KUKA KRL program: MyProgram_139().src

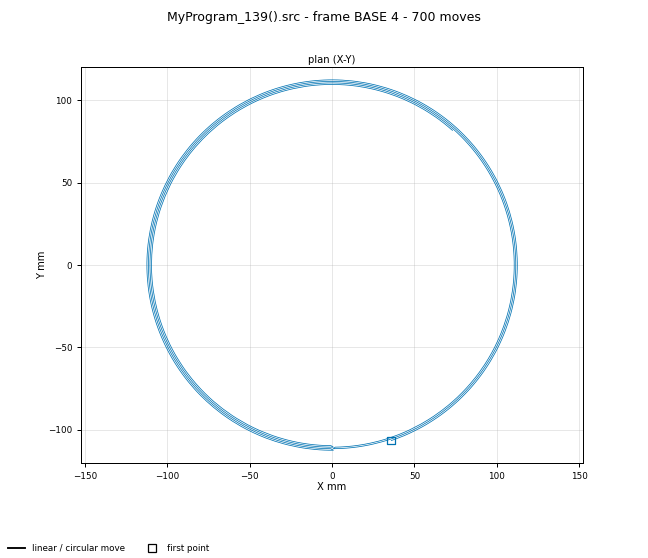
[picture p0: tool path of MyProgram_139().src in frame BASE 4, 700 of 700 moves have a stored position in this frame; points joined in program order, loops and branches not executed]
&ACCESS RVP
&REL 1
&PARAM TEMPLATE = C:\KRC\Roboter\Template\vorgabe
&PARAM EDITMASK = *
DEF MyProgram_139()
; ---- Setting reference (Base) ----
$BASE = BASE_DATA[4]

; --------------------------
; ---- Setting tool (TCP) ----
$TOOL = TOOL_DATA[3]
; --------------------------

$VEL.CP = VEL_APROX_PRINT
Startdeposition()
$VEL.CP = VEL_PRINT
LIN {X 35.9245,Y -106.4874,Z 112,A -74.797,B 24.9523,C -1.5971,E1 25.0523,E2 520.6725} C_DIS
LIN {X 38.4921,Y -105.5865,Z 112,A -73.3956,B 24.9521,C -1.5996,E1 25.056,E2 519.2681} C_DIS
LIN {X 41.1063,Y -104.5964,Z 112,A -71.9841,B 24.952,C -1.6009,E1 25.0597,E2 517.8564} C_DIS
LIN {X 43.6266,Y -103.5706,Z 112,A -70.5551,B 24.9517,C -1.6048,E1 25.0634,E2 516.4215} C_DIS
LIN {X 46.9304,Y -102.1175,Z 112,A -68.8328,B 24.9519,C -1.6024,E1 25.0677,E2 514.7093} C_DIS
LIN {X 49.2943,Y -100.9985,Z 112,A -67.3119,B 24.9513,C -1.6129,E1 25.0716,E2 513.1676} C_DIS
LIN {X 51.7581,Y -99.7583,Z 112,A -66.037,B 24.9515,C -1.6094,E1 25.0748,E2 511.9044} C_DIS
LIN {X 54.1907,Y -98.458,Z 112,A -64.636,B 24.9513,C -1.6116,E1 25.0782,E2 510.5022} C_DIS
LIN {X 56.5907,Y -97.0985,Z 112,A -63.2354,B 24.9512,C -1.6139,E1 25.0816,E2 509.1003} C_DIS
LIN {X 58.9565,Y -95.6804,Z 112,A -61.8347,B 24.951,C -1.6163,E1 25.0849,E2 507.6984} C_DIS
LIN {X 61.2869,Y -94.2047,Z 112,A -60.4345,B 24.9509,C -1.6188,E1 25.0882,E2 506.2969} C_DIS
LIN {X 63.5803,Y -92.6723,Z 112,A -59.034,B 24.9507,C -1.6214,E1 25.0915,E2 504.8951} C_DIS
LIN {X 65.8355,Y -91.0841,Z 112,A -57.6342,B 24.9506,C -1.624,E1 25.0947,E2 503.4939} C_DIS
LIN {X 68.051,Y -89.4409,Z 112,A -56.2343,B 24.9504,C -1.6267,E1 25.0978,E2 502.0926} C_DIS
LIN {X 70.2255,Y -87.744,Z 112,A -54.8346,B 24.9502,C -1.6295,E1 25.1009,E2 500.6916} C_DIS
LIN {X 72.7084,Y -85.6953,Z 112,A -53.1456,B 24.9499,C -1.6354,E1 25.1045,E2 498.995} C_DIS
LIN {X 74.9462,Y -83.7449,Z 112,A -51.6871,B 24.9499,C -1.6364,E1 25.1075,E2 497.54} C_DIS
LIN {X 76.9788,Y -81.8804,Z 112,A -50.292,B 24.9496,C -1.6393,E1 25.1104,E2 496.1439} C_DIS
LIN {X 78.9916,Y -79.9405,Z 112,A -48.8873,B 24.9495,C -1.6418,E1 25.1132,E2 494.7391} C_DIS
LIN {X 81.0209,Y -77.8831,Z 112,A -47.3434,B 24.9491,C -1.6487,E1 25.1162,E2 493.1855} C_DIS
LIN {X 83.2726,Y -75.4738,Z 112,A -45.741,B 24.9491,C -1.6494,E1 25.1192,E2 491.5886} C_DIS
LIN {X 85.0997,Y -73.4075,Z 112,A -44.3426,B 24.9488,C -1.6526,E1 25.1218,E2 490.1888} C_DIS
LIN {X 86.8756,Y -71.2969,Z 112,A -42.9445,B 24.9486,C -1.656,E1 25.1243,E2 488.7891} C_DIS
LIN {X 88.5991,Y -69.1434,Z 112,A -41.5463,B 24.9484,C -1.6594,E1 25.1267,E2 487.3895} C_DIS
LIN {X 90.2693,Y -66.9483,Z 112,A -40.1481,B 24.9482,C -1.6629,E1 25.1291,E2 485.9898} C_DIS
LIN {X 91.8851,Y -64.7128,Z 112,A -38.7504,B 24.948,C -1.6664,E1 25.1313,E2 484.5906} C_DIS
LIN {X 93.4456,Y -62.4383,Z 112,A -37.3524,B 24.9477,C -1.67,E1 25.1335,E2 483.191} C_DIS
LIN {X 94.9497,Y -60.1263,Z 112,A -35.9549,B 24.9475,C -1.6736,E1 25.1356,E2 481.792} C_DIS
LIN {X 96.3967,Y -57.778,Z 112,A -34.5572,B 24.9473,C -1.6773,E1 25.1377,E2 480.3928} C_DIS
LIN {X 97.8454,Y -55.2879,Z 112,A -33.1542,B 24.9472,C -1.6786,E1 25.1396,E2 478.9939} C_DIS
LIN {X 99.1156,Y -52.9784,Z 112,A -31.7626,B 24.9468,C -1.6848,E1 25.1415,E2 477.5951} C_DIS
LIN {X 100.3859,Y -50.53,Z 112,A -30.3653,B 24.9466,C -1.6886,E1 25.1433,E2 476.1962} C_DIS
LIN {X 101.5958,Y -48.0512,Z 112,A -28.9683,B 24.9463,C -1.6924,E1 25.1449,E2 474.7977} C_DIS
LIN {X 102.9129,Y -45.1569,Z 112,A -27.2819,B 24.9458,C -1.7004,E1 25.1469,E2 473.1017} C_DIS
LIN {X 104.0841,Y -42.3868,Z 112,A -25.8344,B 24.9458,C -1.7012,E1 25.1484,E2 471.6602} C_DIS
LIN {X 105.1062,Y -39.7849,Z 112,A -24.4187,B 24.9455,C -1.7052,E1 25.1498,E2 470.243} C_DIS
LIN {X 106.0509,Y -37.1935,Z 112,A -23.0303,B 24.9453,C -1.7088,E1 25.1512,E2 468.8539} C_DIS
LIN {X 106.9203,Y -34.615,Z 112,A -21.6354,B 24.945,C -1.7135,E1 25.1524,E2 467.4558} C_DIS
LIN {X 107.7481,Y -31.945,Z 112,A -20.2283,B 24.9447,C -1.7172,E1 25.1535,E2 466.0479} C_DIS
LIN {X 108.49,Y -29.327,Z 112,A -18.8421,B 24.9445,C -1.7216,E1 25.1545,E2 464.6594} C_DIS
LIN {X 109.1858,Y -26.6196,Z 112,A -17.4437,B 24.9442,C -1.7249,E1 25.1555,E2 463.2612} C_DIS
LIN {X 109.8062,Y -23.932,Z 112,A -16.047,B 24.944,C -1.729,E1 25.1563,E2 461.8631} C_DIS
LIN {X 110.3534,Y -21.2665,Z 112,A -14.6521,B 24.9437,C -1.7338,E1 25.1571,E2 460.4648} C_DIS
LIN {X 110.8421,Y -18.5519,Z 112,A -13.2558,B 24.9434,C -1.7379,E1 25.1578,E2 459.0671} C_DIS
LIN {X 111.264,Y -15.8261,Z 112,A -11.8678,B 24.9432,C -1.7416,E1 25.1583,E2 457.6786} C_DIS
LIN {X 111.6232,Y -13.0539,Z 112,A -10.4525,B 24.9429,C -1.7458,E1 25.1588,E2 456.2617} C_DIS
LIN {X 111.9065,Y -10.3476,Z 112,A -9.0664,B 24.9426,C -1.7503,E1 25.1592,E2 454.8733} C_DIS
LIN {X 112.1268,Y -7.5982,Z 112,A -7.6699,B 24.9423,C -1.7544,E1 25.1595,E2 453.4754} C_DIS
LIN {X 112.2795,Y -4.8441,Z 112,A -6.2383,B 24.9419,C -1.7601,E1 25.1597,E2 452.0387} C_DIS
LIN {X 112.3645,Y -2.0872,Z 112,A -4.844,B 24.9417,C -1.7642,E1 25.1597,E2 450.6432} C_DIS
LIN {X 112.3776,Y 1.3791,Z 112,A -3.1304,B 24.9415,C -1.7674,E1 25.1597,E2 448.9322} C_DIS
LIN {X 112.3099,Y 4.1366,Z 112,A -1.7339,B 24.9412,C -1.7715,E1 25.1597,E2 447.5343} C_DIS
LIN {X 112.1573,Y 7.1466,Z 112,A -0.3253,B 24.9412,C -1.7706,E1 25.1594,E2 446.1362} C_DIS
LIN {X 111.9716,Y 9.6424,Z 112,A 1.0593,B 24.9406,C -1.7797,E1 25.1591,E2 444.7384} C_DIS
LIN {X 111.7013,Y 12.3874,Z 112,A 2.4557,B 24.9404,C -1.7837,E1 25.1587,E2 443.3407} C_DIS
LIN {X 111.3636,Y 15.125,Z 112,A 3.8525,B 24.9401,C -1.7878,E1 25.1582,E2 441.9426} C_DIS
LIN {X 110.9589,Y 17.8534,Z 112,A 5.2493,B 24.9398,C -1.7918,E1 25.1576,E2 440.5445} C_DIS
LIN {X 110.4222,Y 20.9094,Z 112,A 6.9113,B 24.9392,C -1.8005,E1 25.1568,E2 438.8716} C_DIS
LIN {X 109.8062,Y 23.932,Z 112,A 8.3909,B 24.9392,C -1.8012,E1 25.1559,E2 437.3991} C_DIS
LIN {X 109.1858,Y 26.6196,Z 112,A 9.7794,B 24.9389,C -1.8048,E1 25.155,E2 436.0103} C_DIS
LIN {X 108.49,Y 29.327,Z 112,A 11.1865,B 24.9387,C -1.8083,E1 25.154,E2 434.6028} C_DIS
LIN {X 107.7481,Y 31.945,Z 112,A 12.5733,B 24.9384,C -1.8126,E1 25.1529,E2 433.214} C_DIS
LIN {X 106.9203,Y 34.615,Z 112,A 13.9893,B 24.9382,C -1.8165,E1 25.1517,E2 431.7968} C_DIS
LIN {X 106.0509,Y 37.1935,Z 112,A 15.3678,B 24.9379,C -1.8202,E1 25.1505,E2 430.4173} C_DIS
LIN {X 105.1062,Y 39.7849,Z 112,A 16.7649,B 24.9376,C -1.824,E1 25.1491,E2 429.0191} C_DIS
LIN {X 104.0841,Y 42.3868,Z 112,A 18.1727,B 24.9374,C -1.8274,E1 25.1477,E2 427.6111} C_DIS
LIN {X 102.9669,Y 45.0331,Z 112,A 19.7103,B 24.9369,C -1.835,E1 25.1459,E2 426.064} C_DIS
LIN {X 101.4447,Y 48.3656,Z 112,A 21.3327,B 24.9373,C -1.8291,E1 25.1441,E2 424.4642} C_DIS
LIN {X 100.3859,Y 50.53,Z 112,A 22.7141,B 24.9366,C -1.8395,E1 25.1423,E2 423.0656} C_DIS
LIN {X 99.1156,Y 52.9784,Z 112,A 24.1122,B 24.9363,C -1.843,E1 25.1405,E2 421.6666} C_DIS
LIN {X 97.7856,Y 55.3949,Z 112,A 25.5103,B 24.9361,C -1.8465,E1 25.1386,E2 420.2675} C_DIS
LIN {X 96.3967,Y 57.778,Z 112,A 26.9083,B 24.9359,C -1.8499,E1 25.1366,E2 418.8687} C_DIS
LIN {X 94.8065,Y 60.3494,Z 112,A 28.319,B 24.9359,C -1.8481,E1 25.1345,E2 417.4694} C_DIS
LIN {X 93.1455,Y 62.8814,Z 112,A 30.011,B 24.9352,C -1.8588,E1 25.1319,E2 415.7606} C_DIS
LIN {X 91.4738,Y 65.2893,Z 112,A 31.4627,B 24.9352,C -1.8607,E1 25.1296,E2 414.3116} C_DIS
LIN {X 89.8663,Y 67.4848,Z 112,A 32.8425,B 24.9349,C -1.8638,E1 25.1273,E2 412.931} C_DIS
LIN {X 88.16,Y 69.699,Z 112,A 34.2815,B 24.9346,C -1.8679,E1 25.1248,E2 411.4892} C_DIS
LIN {X 85.9941,Y 72.3577,Z 112,A 36.1867,B 24.9338,C -1.879,E1 25.1214,E2 409.5664} C_DIS
LIN {X 83.7449,Y 74.9462,Z 112,A 37.7478,B 24.9341,C -1.8747,E1 25.1185,E2 408.0225} C_DIS
LIN {X 81.8397,Y 77.0221,Z 112,A 39.1555,B 24.934,C -1.8766,E1 25.1158,E2 406.6165} C_DIS
LIN {X 79.9666,Y 78.9651,Z 112,A 40.5704,B 24.9336,C -1.8813,E1 25.1131,E2 405.1964} C_DIS
LIN {X 77.4947,Y 81.3953,Z 112,A 42.298,B 24.9336,C -1.8833,E1 25.1096,E2 403.4715} C_DIS
LIN {X 75.4738,Y 83.2726,Z 112,A 43.698,B 24.9333,C -1.8859,E1 25.1067,E2 402.0711} C_DIS
LIN {X 73.4075,Y 85.0997,Z 112,A 45.0984,B 24.9332,C -1.8884,E1 25.1038,E2 400.6702} C_DIS
LIN {X 71.2969,Y 86.8756,Z 112,A 46.6719,B 24.9324,C -1.8985,E1 25.1004,E2 399.0788} C_DIS
LIN {X 68.6119,Y 89.0087,Z 112,A 48.2399,B 24.9328,C -1.8938,E1 25.0969,E2 397.5278} C_DIS
LIN {X 66.2518,Y 90.7793,Z 112,A 49.8035,B 24.9324,C -1.8991,E1 25.0934,E2 395.9573} C_DIS
LIN {X 63.5804,Y 92.6723,Z 112,A 51.4019,B 24.9324,C -1.8987,E1 25.0898,E2 394.3651} C_DIS
LIN {X 61.2869,Y 94.2047,Z 112,A 52.8033,B 24.9323,C -1.9008,E1 25.0865,E2 392.9636} C_DIS
LIN {X 58.9566,Y 95.6804,Z 112,A 54.2049,B 24.9321,C -1.9027,E1 25.0832,E2 391.5618} C_DIS
LIN {X 56.1014,Y 97.3797,Z 112,A 55.9289,B 24.9319,C -1.9066,E1 25.079,E2 389.8339} C_DIS
LIN {X 53.6009,Y 98.778,Z 112,A 57.3582,B 24.9319,C -1.9073,E1 25.0755,E2 388.4072} C_DIS
LIN {X 51.1606,Y 100.0637,Z 112,A 58.7605,B 24.9317,C -1.9089,E1 25.0721,E2 387.0048} C_DIS
LIN {X 48.656,Y 101.3052,Z 112,A 60.1733,B 24.9316,C -1.9102,E1 25.0685,E2 385.5928} C_DIS
LIN {X 46.1891,Y 102.4535,Z 112,A 61.5571,B 24.9315,C -1.9116,E1 25.065,E2 384.2091} C_DIS
LIN {X 43.5923,Y 103.585,Z 112,A 62.9811,B 24.9315,C -1.9123,E1 25.0613,E2 382.7868} C_DIS
LIN {X 41.1063,Y 104.5964,Z 112,A 64.3632,B 24.9313,C -1.9143,E1 25.0578,E2 381.403} C_DIS
LIN {X 38.527,Y 105.5737,Z 112,A 65.7752,B 24.9312,C -1.9159,E1 25.0541,E2 379.9903} C_DIS
LIN {X 35.9245,Y 106.4874,Z 112,A 67.1702,B 24.9312,C -1.9167,E1 25.0504,E2 378.5964} C_DIS
LIN {X 33.3004,Y 107.337,Z 112,A 68.5826,B 24.931,C -1.918,E1 25.0466,E2 377.1833} C_DIS
LIN {X 30.6204,Y 108.132,Z 112,A 69.9885,B 24.931,C -1.9182,E1 25.0428,E2 375.7793} C_DIS
LIN {X 27.9935,Y 108.8417,Z 112,A 71.3911,B 24.931,C -1.9198,E1 25.0391,E2 374.3753} C_DIS
LIN {X 25.3139,Y 109.4959,Z 112,A 72.787,B 24.9309,C -1.9201,E1 25.0353,E2 372.9806} C_DIS
LIN {X 22.6191,Y 110.0841,Z 112,A 74.2005,B 24.9309,C -1.9211,E1 25.0314,E2 371.5665} C_DIS
LIN {X 19.8741,Y 110.6127,Z 112,A 75.607,B 24.9309,C -1.9209,E1 25.0275,E2 370.1621} C_DIS
LIN {X 17.1536,Y 111.0671,Z 112,A 77.0303,B 24.9307,C -1.922,E1 25.0236,E2 368.7374} C_DIS
LIN {X 14.4596,Y 111.4498,Z 112,A 78.4163,B 24.9307,C -1.9223,E1 25.0198,E2 367.352} C_DIS
LIN {X 11.7201,Y 111.7711,Z 112,A 79.8134,B 24.9307,C -1.9222,E1 25.0159,E2 365.9562} C_DIS
LIN {X 8.9365,Y 112.028,Z 112,A 81.2296,B 24.9307,C -1.9219,E1 25.012,E2 364.5413} C_DIS
LIN {X 6.2216,Y 112.2116,Z 112,A 82.6255,B 24.9307,C -1.9223,E1 25.0081,E2 363.1451} C_DIS
LIN {X 3.4288,Y 112.3316,Z 112,A 84.0425,B 24.9307,C -1.9218,E1 25.0041,E2 361.7297} C_DIS
LIN {X 0.671,Y 112.3819,Z 112,A 85.4492,B 24.9307,C -1.9216,E1 25.0002,E2 360.3236} C_DIS
LIN {X -2.0872,Y 112.3645,Z 112,A 86.8561,B 24.9307,C -1.9213,E1 24.9963,E2 358.9173} C_DIS
LIN {X -4.9758,Y 112.2738,Z 112,A 88.4094,B 24.9306,C -1.9242,E1 24.9919,E2 357.3568} C_DIS
LIN {X -8.2676,Y 112.0815,Z 112,A 90.0218,B 24.9308,C -1.9206,E1 24.9875,E2 355.7524} C_DIS
LIN {X -11.0158,Y 111.8449,Z 112,A 91.4297,B 24.9308,C -1.92,E1 24.9835,E2 354.3453} C_DIS
LIN {X -13.7572,Y 111.5408,Z 112,A 92.8377,B 24.9309,C -1.9192,E1 24.9796,E2 352.9381} C_DIS
LIN {X -16.4905,Y 111.1696,Z 112,A 94.2457,B 24.931,C -1.9184,E1 24.9758,E2 351.531} C_DIS
LIN {X -19.2137,Y 110.7314,Z 112,A 95.7178,B 24.9309,C -1.9201,E1 24.9717,E2 350.0534} C_DIS
LIN {X -21.9254,Y 110.2266,Z 112,A 97.063,B 24.9311,C -1.9164,E1 24.968,E2 348.7154} C_DIS
LIN {X -24.6239,Y 109.6553,Z 112,A 98.5972,B 24.9309,C -1.9205,E1 24.9638,E2 347.1697} C_DIS
LIN {X -27.3076,Y 109.018,Z 112,A 99.8811,B 24.9313,C -1.9141,E1 24.9604,E2 345.8992} C_DIS
LIN {X -29.9748,Y 108.315,Z 112,A 101.2904,B 24.9314,C -1.9128,E1 24.9566,E2 344.4909} C_DIS
LIN {X -32.6239,Y 107.5467,Z 112,A 102.7001,B 24.9315,C -1.9113,E1 24.9528,E2 343.0823} C_DIS
LIN {X -35.2534,Y 106.7137,Z 112,A 104.2715,B 24.9311,C -1.9165,E1 24.9486,E2 341.4958} C_DIS
LIN {X -38.4921,Y 105.5865,Z 112,A 105.863,B 24.9318,C -1.9078,E1 24.9444,E2 339.9216} C_DIS
LIN {X -41.0717,Y 104.61,Z 112,A 107.2734,B 24.9318,C -1.9061,E1 24.9408,E2 338.5123} C_DIS
LIN {X -43.6266,Y 103.5706,Z 112,A 108.6925,B 24.932,C -1.9046,E1 24.9371,E2 337.0935} C_DIS
LIN {X -46.1891,Y 102.4535,Z 112,A 110.1051,B 24.9322,C -1.902,E1 24.9335,E2 335.6838} C_DIS
LIN {X -48.656,Y 101.3052,Z 112,A 111.5057,B 24.9322,C -1.9004,E1 24.93,E2 334.2835} C_DIS
LIN {X -51.1606,Y 100.0637,Z 112,A 112.9272,B 24.9325,C -1.8979,E1 24.9264,E2 332.8641} C_DIS
LIN {X -53.6009,Y 98.778,Z 112,A 114.3388,B 24.9326,C -1.8957,E1 24.923,E2 331.4537} C_DIS
LIN {X -55.9767,Y 97.4513,Z 112,A 115.7602,B 24.9327,C -1.8946,E1 24.9195,E2 330.0307} C_DIS
LIN {X -58.3831,Y 96.0289,Z 112,A 117.1708,B 24.9329,C -1.8914,E1 24.9161,E2 328.6234} C_DIS
LIN {X -60.7222,Y 94.5672,Z 112,A 118.5742,B 24.9331,C -1.8887,E1 24.9128,E2 327.2222} C_DIS
LIN {X -62.9939,Y 93.0694,Z 112,A 119.9761,B 24.9333,C -1.8865,E1 24.9096,E2 325.8207} C_DIS
LIN {X -65.259,Y 91.4954,Z 112,A 121.4182,B 24.9333,C -1.8851,E1 24.9063,E2 324.377} C_DIS
LIN {X -68.051,Y 89.4409,Z 112,A 123.1639,B 24.9337,C -1.8805,E1 24.9024,E2 322.636} C_DIS
LIN {X -70.2255,Y 87.744,Z 112,A 124.5768,B 24.9339,C -1.8777,E1 24.8993,E2 321.2246} C_DIS
LIN {X -72.3577,Y 85.9941,Z 112,A 125.9898,B 24.9341,C -1.8749,E1 24.8963,E2 319.8129} C_DIS
LIN {X -74.4463,Y 84.1925,Z 112,A 127.4029,B 24.9343,C -1.8719,E1 24.8933,E2 318.4013} C_DIS
LIN {X -76.49,Y 82.3401,Z 112,A 128.8558,B 24.9344,C -1.8705,E1 24.8903,E2 316.9458} C_DIS
LIN {X -78.4877,Y 80.4381,Z 112,A 130.2301,B 24.9347,C -1.8659,E1 24.8875,E2 315.5769} C_DIS
LIN {X -80.4381,Y 78.4877,Z 112,A 131.6436,B 24.935,C -1.8627,E1 24.8848,E2 314.1649} C_DIS
LIN {X -82.3401,Y 76.49,Z 112,A 133.1357,B 24.935,C -1.8627,E1 24.8819,E2 312.6665} C_DIS
LIN {X -84.1925,Y 74.4463,Z 112,A 134.6402,B 24.935,C -1.8629,E1 24.8791,E2 311.1546} C_DIS
LIN {X -86.423,Y 71.8416,Z 112,A 136.2294,B 24.9357,C -1.8521,E1 24.8763,E2 309.5839} C_DIS
LIN {X -88.16,Y 69.699,Z 112,A 137.6526,B 24.9359,C -1.849,E1 24.8738,E2 308.1613} C_DIS
LIN {X -89.8663,Y 67.4848,Z 112,A 139.0688,B 24.9362,C -1.8448,E1 24.8714,E2 306.7483} C_DIS
LIN {X -91.4738,Y 65.2893,Z 112,A 140.473,B 24.9364,C -1.8417,E1 24.8691,E2 305.3448} C_DIS
LIN {X -93.0485,Y 63.0247,Z 112,A 141.8877,B 24.9367,C -1.8381,E1 24.8669,E2 303.9316} C_DIS
LIN {X -94.5672,Y 60.7222,Z 112,A 143.3025,B 24.9369,C -1.8345,E1 24.8647,E2 302.5183} C_DIS
LIN {X -96.0482,Y 58.3514,Z 112,A 144.7368,B 24.9372,C -1.8308,E1 24.8626,E2 301.0856} C_DIS
LIN {X -97.4328,Y 56.0089,Z 112,A 146.1434,B 24.9374,C -1.8275,E1 24.8607,E2 299.6795} C_DIS
LIN {X -98.778,Y 53.6009,Z 112,A 147.5478,B 24.9377,C -1.8233,E1 24.8588,E2 298.2777} C_DIS
LIN {X -100.0806,Y 51.1275,Z 112,A 148.9824,B 24.938,C -1.8194,E1 24.8569,E2 296.8446} C_DIS
LIN {X -101.2891,Y 48.6895,Z 112,A 150.3871,B 24.9382,C -1.816,E1 24.8552,E2 295.4406} C_DIS
LIN {X -102.4687,Y 46.1552,Z 112,A 151.8132,B 24.9385,C -1.8117,E1 24.8536,E2 294.0169} C_DIS
LIN {X -103.5561,Y 43.6609,Z 112,A 153.2607,B 24.9386,C -1.8098,E1 24.852,E2 292.5659} C_DIS
LIN {X -104.8554,Y 40.4472,Z 112,A 154.9888,B 24.9391,C -1.8028,E1 24.8502,E2 290.8449} C_DIS
LIN {X -105.8164,Y 37.8617,Z 112,A 156.4047,B 24.9394,C -1.7988,E1 24.8488,E2 289.4305} C_DIS
LIN {X -106.7137,Y 35.2534,Z 112,A 157.8204,B 24.9396,C -1.7947,E1 24.8476,E2 288.0164} C_DIS
LIN {X -107.5467,Y 32.6239,Z 112,A 159.2363,B 24.9399,C -1.7907,E1 24.8464,E2 286.602} C_DIS
LIN {X -108.315,Y 29.9748,Z 112,A 160.8138,B 24.9398,C -1.7929,E1 24.8452,E2 285.01} C_DIS
LIN {X -109.1858,Y 26.6196,Z 112,A 162.423,B 24.9405,C -1.7811,E1 24.8441,E2 283.4196} C_DIS
LIN {X -109.7983,Y 23.9683,Z 112,A 163.8288,B 24.9408,C -1.7774,E1 24.8433,E2 282.0144} C_DIS
LIN {X -110.3534,Y 21.2665,Z 112,A 165.2535,B 24.941,C -1.7736,E1 24.8425,E2 280.5903} C_DIS
LIN {X -110.8482,Y 18.5152,Z 112,A 166.6799,B 24.9413,C -1.769,E1 24.8418,E2 279.1664} C_DIS
LIN {X -111.264,Y 15.8261,Z 112,A 168.1295,B 24.9415,C -1.767,E1 24.8412,E2 277.713} C_DIS
LIN {X -111.7013,Y 12.3874,Z 112,A 169.8567,B 24.942,C -1.7597,E1 24.8407,E2 275.9929} C_DIS
LIN {X -111.9716,Y 9.6424,Z 112,A 171.273,B 24.9422,C -1.7555,E1 24.8403,E2 274.5781} C_DIS
LIN {X -112.1745,Y 6.8916,Z 112,A 172.689,B 24.9425,C -1.7513,E1 24.84,E2 273.1635} C_DIS
LIN {X -112.3099,Y 4.1366,Z 112,A 174.2199,B 24.9425,C -1.7516,E1 24.8398,E2 271.6227} C_DIS
LIN {X -112.3776,Y 1.3791,Z 112,A 175.6197,B 24.9428,C -1.7468,E1 24.8398,E2 270.2259} C_DIS
LIN {X -112.3645,Y -2.0872,Z 112,A 177.2923,B 24.9434,C -1.7374,E1 24.8398,E2 268.5656} C_DIS
LIN {X -112.2795,Y -4.8441,Z 112,A 178.7083,B 24.9437,C -1.7332,E1 24.84,E2 267.151} C_DIS
LIN {X -112.1268,Y -7.5982,Z 112,A -179.8754,B 24.944,C -1.7291,E1 24.8402,E2 265.7361} C_DIS
LIN {X -111.9065,Y -10.3476,Z 112,A -178.4596,B 24.9442,C -1.725,E1 24.8406,E2 264.3216} C_DIS
LIN {X -111.6232,Y -13.0539,Z 112,A -177.0452,B 24.9445,C -1.7216,E1 24.841,E2 262.9068} C_DIS
LIN {X -111.264,Y -15.8261,Z 112,A -175.6275,B 24.9448,C -1.7168,E1 24.8415,E2 261.4922} C_DIS
LIN {X -110.8421,Y -18.5519,Z 112,A -174.2114,B 24.945,C -1.7127,E1 24.8422,E2 260.0773} C_DIS
LIN {X -110.3534,Y -21.2665,Z 112,A -172.7871,B 24.9453,C -1.709,E1 24.8429,E2 258.6534} C_DIS
LIN {X -109.7388,Y -24.241,Z 112,A -171.1876,B 24.9454,C -1.7061,E1 24.8438,E2 257.0513} C_DIS
LIN {X -109.018,Y -27.3076,Z 112,A -169.6111,B 24.9458,C -1.7,E1 24.8449,E2 255.4803} C_DIS
LIN {X -108.315,Y -29.9748,Z 112,A -168.1956,B 24.9461,C -1.696,E1 24.8459,E2 254.066} C_DIS
LIN {X -107.5467,Y -32.6239,Z 112,A -166.78,B 24.9463,C -1.6921,E1 24.847,E2 252.6515} C_DIS
LIN {X -106.7137,Y -35.2534,Z 112,A -165.3645,B 24.9466,C -1.6882,E1 24.8482,E2 251.2372} C_DIS
LIN {X -105.8164,Y -37.8617,Z 112,A -163.9492,B 24.9468,C -1.6844,E1 24.8495,E2 249.823} C_DIS
LIN {X -104.8554,Y -40.4472,Z 112,A -162.3656,B 24.9467,C -1.6873,E1 24.8511,E2 248.2236} C_DIS
LIN {X -103.5706,Y -43.6266,Z 112,A -160.7746,B 24.9474,C -1.676,E1 24.8528,E2 246.6507} C_DIS
LIN {X -102.4535,Y -46.1891,Z 112,A -159.3404,B 24.9476,C -1.6722,E1 24.8544,E2 245.2175} C_DIS
LIN {X -101.2891,Y -48.6895,Z 112,A -157.903,B 24.9478,C -1.6695,E1 24.8562,E2 243.7788} C_DIS
LIN {X -99.7583,Y -51.7581,Z 112,A -156.1667,B 24.9481,C -1.6641,E1 24.8583,E2 242.0461} C_DIS
LIN {X -98.458,Y -54.1907,Z 112,A -154.7521,B 24.9483,C -1.6606,E1 24.8602,E2 240.6324} C_DIS
LIN {X -97.0985,Y -56.5907,Z 112,A -153.2799,B 24.9483,C -1.6594,E1 24.8623,E2 239.1553} C_DIS
LIN {X -95.6804,Y -58.9565,Z 112,A -151.9233,B 24.9488,C -1.6537,E1 24.8643,E2 237.8054} C_DIS
LIN {X -94.2047,Y -61.2869,Z 112,A -150.383,B 24.9486,C -1.6554,E1 24.8666,E2 236.2533} C_DIS
LIN {X -92.6723,Y -63.5803,Z 112,A -148.9587,B 24.9488,C -1.6525,E1 24.8688,E2 234.8287} C_DIS
LIN {X -90.6877,Y -66.3769,Z 112,A -147.3288,B 24.9494,C -1.6434,E1 24.8715,E2 233.2125} C_DIS
LIN {X -89.0087,Y -68.6119,Z 112,A -145.9134,B 24.9496,C -1.6396,E1 24.8739,E2 231.7996} C_DIS
LIN {X -87.2981,Y -70.7756,Z 112,A -144.4909,B 24.9498,C -1.6368,E1 24.8763,E2 230.3769} C_DIS
LIN {X -85.5348,Y -72.8967,Z 112,A -143.0863,B 24.95,C -1.6335,E1 24.8789,E2 228.9739} C_DIS
LIN {X -83.7449,Y -74.9462,Z 112,A -141.675,B 24.9501,C -1.6313,E1 24.8815,E2 227.5614} C_DIS
LIN {X -81.8804,Y -76.9788,Z 112,A -140.2705,B 24.9503,C -1.6281,E1 24.8842,E2 226.1584} C_DIS
LIN {X -79.9405,Y -78.9916,Z 112,A -138.8473,B 24.9505,C -1.6249,E1 24.8869,E2 224.7366} C_DIS
LIN {X -77.9778,Y -80.9296,Z 112,A -137.4261,B 24.9507,C -1.6226,E1 24.8898,E2 223.315} C_DIS
LIN {X -75.9956,Y -82.7938,Z 112,A -136.0239,B 24.9508,C -1.6204,E1 24.8926,E2 221.9125} C_DIS
LIN {X -73.9129,Y -84.6583,Z 112,A -134.61,B 24.951,C -1.6171,E1 24.8956,E2 220.5007} C_DIS
LIN {X -71.8416,Y -86.423,Z 112,A -133.181,B 24.951,C -1.6161,E1 24.8987,E2 219.0685} C_DIS
LIN {X -69.6699,Y -88.1831,Z 112,A -131.7637,B 24.9512,C -1.6132,E1 24.9017,E2 217.6529} C_DIS
LIN {X -67.5145,Y -89.844,Z 112,A -130.376,B 24.9514,C -1.6107,E1 24.9048,E2 216.2661} C_DIS
LIN {X -65.1106,Y -91.6013,Z 112,A -128.8017,B 24.9514,C -1.6104,E1 24.9084,E2 214.687} C_DIS
LIN {X -62.4383,Y -93.4456,Z 112,A -127.1995,B 24.9517,C -1.6055,E1 24.9121,E2 213.0911} C_DIS
LIN {X -60.1263,Y -94.9497,Z 112,A -125.7887,B 24.9518,C -1.6035,E1 24.9154,E2 211.6805} C_DIS
LIN {X -57.6584,Y -96.4674,Z 112,A -124.3714,B 24.9521,C -1.5989,E1 24.9188,E2 210.2699} C_DIS
LIN {X -55.3949,Y -97.7856,Z 112,A -122.9674,B 24.9521,C -1.5998,E1 24.9222,E2 208.8596} C_DIS
LIN {X -52.9784,Y -99.1156,Z 112,A -121.5571,B 24.9521,C -1.5981,E1 24.9257,E2 207.4493} C_DIS
LIN {X -50.376,Y -100.4623,Z 112,A -120.1388,B 24.9524,C -1.593,E1 24.9292,E2 206.0392} C_DIS
LIN {X -47.5702,Y -101.8197,Z 112,A -118.4297,B 24.9523,C -1.5962,E1 24.9335,E2 204.3183} C_DIS
LIN {X -44.8943,Y -103.0274,Z 112,A -116.9656,B 24.9524,C -1.5932,E1 24.9372,E2 202.8579} C_DIS
LIN {X -42.3868,Y -104.0841,Z 112,A -115.5752,B 24.9525,C -1.5919,E1 24.9408,E2 201.4674} C_DIS
LIN {X -39.7849,Y -105.1062,Z 112,A -114.1472,B 24.9525,C -1.5906,E1 24.9445,E2 200.0392} C_DIS
LIN {X -37.1935,Y -106.0509,Z 112,A -112.7467,B 24.9527,C -1.5891,E1 24.9482,E2 198.6395} C_DIS
LIN {X -34.615,Y -106.9203,Z 112,A -111.34,B 24.9527,C -1.5889,E1 24.952,E2 197.2309} C_DIS
LIN {X -31.945,Y -107.7481,Z 112,A -109.921,B 24.9527,C -1.5876,E1 24.9557,E2 195.8125} C_DIS
LIN {X -29.327,Y -108.49,Z 112,A -108.5234,B 24.9528,C -1.5871,E1 24.9595,E2 194.4138} C_DIS
LIN {X -26.6196,Y -109.1858,Z 112,A -107.1136,B 24.9528,C -1.5857,E1 24.9633,E2 193.0055} C_DIS
LIN {X -23.932,Y -109.8062,Z 112,A -105.7058,B 24.9529,C -1.5851,E1 24.9672,E2 191.5974} C_DIS
LIN {X -21.2665,Y -110.3534,Z 112,A -104.3,B 24.9529,C -1.5853,E1 24.971,E2 190.1894} C_DIS
LIN {X -18.5519,Y -110.8421,Z 112,A -102.893,B 24.9529,C -1.5849,E1 24.9749,E2 188.782} C_DIS
LIN {X -15.8261,Y -111.264,Z 112,A -101.4946,B 24.9529,C -1.5842,E1 24.9788,E2 187.3841} C_DIS
LIN {X -13.0539,Y -111.6232,Z 112,A -100.0688,B 24.9529,C -1.584,E1 24.9827,E2 185.9578} C_DIS
LIN {X -10.3476,Y -111.9065,Z 112,A -98.6727,B 24.9529,C -1.5842,E1 24.9866,E2 184.5604} C_DIS
LIN {X -7.5982,Y -112.1268,Z 112,A -97.2665,B 24.9529,C -1.5842,E1 24.9905,E2 183.1536} C_DIS
LIN {X -4.8441,Y -112.2795,Z 112,A -95.8604,B 24.9529,C -1.5843,E1 24.9944,E2 181.7469} C_DIS
LIN {X -2.0872,Y -112.3645,Z 112,A -94.4546,B 24.9529,C -1.5845,E1 24.9984,E2 180.3405} C_DIS
LIN {X 0.7859,Y -112.3805,Z 112,A -93.0437,B 24.9531,C -1.5825,E1 25.0023,E2 178.9343} C_DIS
Enddeposition()
LIN {X 0.7859,Y -112.3805,Z 112,A -93.0437,B 24.9531,C -1.5825,E1 25.0023,E2 178.9343} C_DIS
Startdeposition()
$VEL.CP = VEL_PRINT
LIN {X -0.7886,Y -111.4503,Z 112,A -94.532,B 24.9538,C -1.5696,E1 24.998,E2 180.4531} C_DIS
LIN {X -4.301,Y -111.3711,Z 112,A -96.4382,B 24.9541,C -1.5652,E1 24.9927,E2 182.3702} C_DIS
LIN {X -7.7857,Y -111.1811,Z 112,A -98.2597,B 24.9541,C -1.564,E1 24.9876,E2 184.1951} C_DIS
LIN {X -11.7058,Y -110.8367,Z 112,A -100.0896,B 24.9537,C -1.5722,E1 24.9826,E2 186.0065} C_DIS
LIN {X -14.6972,Y -110.4804,Z 112,A -101.7245,B 24.9539,C -1.5689,E1 24.978,E2 187.6504} C_DIS
LIN {X -18.2607,Y -109.947,Z 112,A -103.5992,B 24.9539,C -1.5685,E1 24.9728,E2 189.5278} C_DIS
LIN {X -21.7585,Y -109.3105,Z 112,A -105.5598,B 24.9542,C -1.5636,E1 24.9674,E2 191.502} C_DIS
LIN {X -25.5515,Y -108.4856,Z 112,A -107.4472,B 24.9539,C -1.5691,E1 24.9623,E2 193.3789} C_DIS
LIN {X -29.0377,Y -107.6039,Z 112,A -109.3211,B 24.9539,C -1.5691,E1 24.9572,E2 195.2554} C_DIS
LIN {X -33.0849,Y -106.4292,Z 112,A -111.3908,B 24.9535,C -1.5747,E1 24.9517,E2 197.3154} C_DIS
LIN {X -36.6323,Y -105.2613,Z 112,A -113.3638,B 24.9535,C -1.5741,E1 24.9465,E2 199.2937} C_DIS
LIN {X -39.9123,Y -104.0625,Z 112,A -115.2052,B 24.9535,C -1.5738,E1 24.9417,E2 201.1394} C_DIS
LIN {X -45.1062,Y -101.9195,Z 112,A -117.9023,B 24.953,C -1.5846,E1 24.9348,E2 203.817} C_DIS
LIN {X -48.7711,Y -100.2171,Z 112,A -120.3822,B 24.9538,C -1.5708,E1 24.9284,E2 206.3361} C_DIS
LIN {X -52.9138,Y -98.0917,Z 112,A -122.5772,B 24.9531,C -1.5819,E1 24.923,E2 208.5107} C_DIS
LIN {X -56.4237,Y -96.1159,Z 112,A -124.6492,B 24.9529,C -1.5848,E1 24.918,E2 210.582} C_DIS
LIN {X -60.2335,Y -93.7748,Z 112,A -126.8739,B 24.9526,C -1.5913,E1 24.9128,E2 212.7982} C_DIS
LIN {X -63.1932,Y -91.8078,Z 112,A -128.9307,B 24.9529,C -1.5851,E1 24.908,E2 214.8768} C_DIS
LIN {X -66.0392,Y -89.7812,Z 112,A -130.55,B 24.9523,C -1.5952,E1 24.9044,E2 216.4776} C_DIS
LIN {X -69.014,Y -87.5149,Z 112,A -132.5091,B 24.9522,C -1.5972,E1 24.9,E2 218.439} C_DIS
LIN {X -72.1359,Y -84.9601,Z 112,A -134.4072,B 24.9515,C -1.6082,E1 24.896,E2 220.3184} C_DIS
LIN {X -74.2883,Y -83.0845,Z 112,A -136.0341,B 24.9517,C -1.6047,E1 24.8925,E2 221.9599} C_DIS
LIN {X -76.8269,Y -80.7451,Z 112,A -137.8654,B 24.9517,C -1.6061,E1 24.8888,E2 223.7955} C_DIS
LIN {X -79.342,Y -78.2728,Z 112,A -139.6433,B 24.9513,C -1.6114,E1 24.8853,E2 225.5683} C_DIS
LIN {X -82.4055,Y -75.0419,Z 112,A -141.8457,B 24.9508,C -1.6198,E1 24.8811,E2 227.7602} C_DIS
LIN {X -84.3423,Y -72.8597,Z 112,A -143.4665,B 24.9509,C -1.6185,E1 24.8781,E2 229.3915} C_DIS
LIN {X -86.4967,Y -70.286,Z 112,A -145.182,B 24.9506,C -1.623,E1 24.8751,E2 231.1043} C_DIS
LIN {X -88.5986,Y -67.6191,Z 112,A -147.1859,B 24.951,C -1.6171,E1 24.8716,E2 233.1316} C_DIS
LIN {X -91.5343,Y -63.5866,Z 112,A -149.4663,B 24.9499,C -1.6346,E1 24.868,E2 235.3814} C_DIS
LIN {X -93.51,Y -60.6461,Z 112,A -151.705,B 24.9506,C -1.6231,E1 24.8645,E2 237.6589} C_DIS
LIN {X -95.6435,Y -57.2228,Z 112,A -153.4984,B 24.9496,C -1.6394,E1 24.8619,E2 239.4225} C_DIS
LIN {X -97.437,Y -54.1099,Z 112,A -155.3242,B 24.9493,C -1.6453,E1 24.8594,E2 241.2439} C_DIS
LIN {X -99.4741,Y -50.2686,Z 112,A -157.4554,B 24.9486,C -1.6555,E1 24.8567,E2 243.3621} C_DIS
LIN {X -102.1615,Y -44.5511,Z 112,A -160.7653,B 24.9482,C -1.6624,E1 24.8528,E2 246.6738} C_DIS
LIN {X -103.3461,Y -41.7309,Z 112,A -162.2777,B 24.9478,C -1.6692,E1 24.8512,E2 248.1782} C_DIS
LIN {X -104.4099,Y -38.9951,Z 112,A -163.9796,B 24.948,C -1.6662,E1 24.8495,E2 249.8968} C_DIS
LIN {X -105.5974,Y -35.6506,Z 112,A -165.6825,B 24.9473,C -1.6764,E1 24.8479,E2 251.5852} C_DIS
LIN {X -106.5131,Y -32.8143,Z 112,A -167.3596,B 24.9473,C -1.6755,E1 24.8465,E2 253.2742} C_DIS
LIN {X -107.7447,Y -28.5165,Z 112,A -169.4575,B 24.9465,C -1.6902,E1 24.845,E2 255.3491} C_DIS
LIN {X -108.8974,Y -23.7307,Z 112,A -171.9333,B 24.9458,C -1.7001,E1 24.8434,E2 257.8157} C_DIS
LIN {X -109.4671,Y -20.9462,Z 112,A -173.625,B 24.9461,C -1.6959,E1 24.8424,E2 259.5275} C_DIS
LIN {X -110.1328,Y -17.1039,Z 112,A -175.7226,B 24.9459,C -1.6987,E1 24.8415,E2 261.631} C_DIS
LIN {X -110.6237,Y -13.5858,Z 112,A -177.4896,B 24.9454,C -1.7067,E1 24.8408,E2 263.3893} C_DIS
LIN {X -110.9633,Y -10.4386,Z 112,A -179.0974,B 24.945,C -1.7127,E1 24.8404,E2 264.9926} C_DIS
LIN {X -111.218,Y -7.2402,Z 112,A 179.2726,B 24.9446,C -1.7187,E1 24.8401,E2 266.618} C_DIS
LIN {X -111.3872,Y -3.854,Z 112,A 177.4088,B 24.9446,C -1.7197,E1 24.8398,E2 268.4905} C_DIS
LIN {X -111.4548,Y -0.1917,Z 112,A 175.4328,B 24.9444,C -1.7223,E1 24.8398,E2 270.4724} C_DIS
LIN {X -111.3916,Y 3.7103,Z 112,A 173.4705,B 24.9439,C -1.7305,E1 24.8399,E2 272.4269} C_DIS
LIN {X -111.2085,Y 7.3809,Z 112,A 171.5514,B 24.9436,C -1.7355,E1 24.8402,E2 274.3456} C_DIS
LIN {X -110.8596,Y 11.4864,Z 112,A 169.4584,B 24.943,C -1.7433,E1 24.8408,E2 276.4325} C_DIS
LIN {X -110.3416,Y 15.7004,Z 112,A 167.3503,B 24.9424,C -1.7532,E1 24.8415,E2 278.5296} C_DIS
LIN {X -109.8397,Y 18.9023,Z 112,A 165.5593,B 24.9424,C -1.7538,E1 24.8424,E2 280.3298} C_DIS
LIN {X -108.9905,Y 23.3038,Z 112,A 163.5025,B 24.9412,C -1.7707,E1 24.8435,E2 282.3585} C_DIS
LIN {X -108.0971,Y 27.1509,Z 112,A 161.1465,B 24.9416,C -1.7648,E1 24.845,E2 284.7425} C_DIS
LIN {X -106.3199,Y 33.4375,Z 112,A 157.818,B 24.9408,C -1.7766,E1 24.8476,E2 288.0622} C_DIS
LIN {X -105.0888,Y 37.1238,Z 112,A 155.6531,B 24.9408,C -1.7765,E1 24.8496,E2 290.2396} C_DIS
LIN {X -103.522,Y 41.2954,Z 112,A 153.5393,B 24.9399,C -1.7903,E1 24.8517,E2 292.3323} C_DIS
LIN {X -102.1811,Y 44.5062,Z 112,A 151.7739,B 24.9395,C -1.7967,E1 24.8536,E2 294.0922} C_DIS
LIN {X -100.6271,Y 47.9178,Z 112,A 149.7071,B 24.9395,C -1.7971,E1 24.8561,E2 296.1691} C_DIS
LIN {X -97.7238,Y 53.5921,Z 112,A 146.6276,B 24.9383,C -1.8144,E1 24.86,E2 299.224} C_DIS
LIN {X -96.1402,Y 56.3826,Z 112,A 145.0955,B 24.9377,C -1.8237,E1 24.8621,E2 300.7418} C_DIS
LIN {X -94.5265,Y 59.0467,Z 112,A 143.3059,B 24.9378,C -1.8211,E1 24.8648,E2 302.5469} C_DIS
LIN {X -91.3559,Y 63.8433,Z 112,A 140.3493,B 24.9373,C -1.8293,E1 24.8694,E2 305.4986} C_DIS
LIN {X -87.9081,Y 68.5151,Z 112,A 137.0922,B 24.9374,C -1.8269,E1 24.8749,E2 308.7771} C_DIS
LIN {X -84.4379,Y 72.749,Z 112,A 134.5388,B 24.9362,C -1.8443,E1 24.8794,E2 311.3008} C_DIS
LIN {X -82.291,Y 75.1667,Z 112,A 132.7733,B 24.9362,C -1.8446,E1 24.8827,E2 313.0735} C_DIS
LIN {X -79.974,Y 77.628,Z 112,A 130.8481,B 24.9364,C -1.8416,E1 24.8864,E2 315.0141} C_DIS
LIN {X -76.4107,Y 81.1369,Z 112,A 128.45,B 24.9355,C -1.8545,E1 24.8912,E2 317.3915} C_DIS
LIN {X -74.1613,Y 83.1982,Z 112,A 126.9597,B 24.9351,C -1.8611,E1 24.8943,E2 318.8719} C_DIS
LIN {X -72.1219,Y 84.9721,Z 112,A 125.5446,B 24.9349,C -1.8633,E1 24.8973,E2 320.2874} C_DIS
LIN {X -69.3635,Y 87.2387,Z 112,A 123.3271,B 24.9357,C -1.8524,E1 24.9022,E2 322.5391} C_DIS
LIN {X -66.4222,Y 89.5002,Z 112,A 121.5922,B 24.9349,C -1.8631,E1 24.906,E2 324.2548} C_DIS
LIN {X -63.4534,Y 91.6269,Z 112,A 119.8874,B 24.9342,C -1.8737,E1 24.9098,E2 325.9403} C_DIS
LIN {X -58.5652,Y 94.8273,Z 112,A 116.8918,B 24.9338,C -1.8797,E1 24.9169,E2 328.9312} C_DIS
LIN {X -55.6655,Y 96.5565,Z 112,A 114.8909,B 24.9343,C -1.8725,E1 24.9217,E2 330.9553} C_DIS
LIN {X -51.9656,Y 98.5969,Z 112,A 112.9138,B 24.9335,C -1.8839,E1 24.9265,E2 332.911} C_DIS
LIN {X -48.937,Y 100.1366,Z 112,A 110.8252,B 24.9342,C -1.8732,E1 24.9319,E2 335.0305} C_DIS
LIN {X -45.2623,Y 101.8501,Z 112,A 108.9821,B 24.9333,C -1.8858,E1 24.9365,E2 336.8479} C_DIS
LIN {X -41.8096,Y 103.314,Z 112,A 107.1617,B 24.9328,C -1.8929,E1 24.9411,E2 338.6557} C_DIS
LIN {X -38.7294,Y 104.5091,Z 112,A 105.3097,B 24.9331,C -1.889,E1 24.946,E2 340.5208} C_DIS
LIN {X -35.234,Y 105.7379,Z 112,A 103.2844,B 24.9333,C -1.8866,E1 24.9514,E2 342.5558} C_DIS
LIN {X -31.7247,Y 106.8425,Z 112,A 101.5561,B 24.9327,C -1.8952,E1 24.956,E2 344.2665} C_DIS
LIN {X -27.731,Y 107.948,Z 112,A 99.518,B 24.9322,C -1.9011,E1 24.9614,E2 346.2936} C_DIS
LIN {X -24.2898,Y 108.7754,Z 112,A 97.5423,B 24.9326,C -1.8965,E1 24.9668,E2 348.2829} C_DIS
LIN {X -20.7824,Y 109.4987,Z 112,A 95.8544,B 24.932,C -1.9042,E1 24.9714,E2 349.9545} C_DIS
LIN {X -16.5694,Y 110.2155,Z 112,A 93.5057,B 24.9324,C -1.8996,E1 24.9779,E2 352.3162} C_DIS
LIN {X -12.7823,Y 110.7178,Z 112,A 91.6639,B 24.9319,C -1.9057,E1 24.983,E2 354.1447} C_DIS
LIN {X -9.1413,Y 111.0778,Z 112,A 89.753,B 24.9319,C -1.9054,E1 24.9883,E2 356.0573} C_DIS
LIN {X -5.8479,Y 111.2999,Z 112,A 87.9898,B 24.9321,C -1.9034,E1 24.9932,E2 357.8259} C_DIS
LIN {X -1.9691,Y 111.4357,Z 112,A 86.0883,B 24.9318,C -1.9078,E1 24.9985,E2 359.7172} C_DIS
LIN {X 1.4591,Y 111.4451,Z 112,A 84.2445,B 24.932,C -1.9047,E1 25.0037,E2 361.5681} C_DIS
LIN {X 5.0011,Y 111.341,Z 112,A 82.4274,B 24.932,C -1.9051,E1 25.0088,E2 363.384} C_DIS
LIN {X 8.9479,Y 111.0933,Z 112,A 80.4522,B 24.9318,C -1.9074,E1 25.0142,E2 365.3527} C_DIS
LIN {X 12.4723,Y 110.7541,Z 112,A 78.5453,B 24.9321,C -1.9035,E1 25.0196,E2 367.2676} C_DIS
LIN {X 16.0044,Y 110.2985,Z 112,A 76.7963,B 24.9319,C -1.9065,E1 25.0244,E2 369.008} C_DIS
LIN {X 19.5282,Y 109.7291,Z 112,A 74.9547,B 24.9319,C -1.9056,E1 25.0294,E2 370.8499} C_DIS
LIN {X 22.9019,Y 109.0758,Z 112,A 73.1854,B 24.9319,C -1.9047,E1 25.0343,E2 372.6192} C_DIS
LIN {X 26.2651,Y 108.3141,Z 112,A 71.434,B 24.9319,C -1.9047,E1 25.039,E2 374.3683} C_DIS
LIN {X 29.3286,Y 107.5253,Z 112,A 69.7262,B 24.9323,C -1.9001,E1 25.0437,E2 376.084} C_DIS
LIN {X 33.7378,Y 106.2257,Z 112,A 67.3483,B 24.9325,C -1.8977,E1 25.05,E2 378.4634} C_DIS
LIN {X 37.1734,Y 105.0714,Z 112,A 64.8036,B 24.9346,C -1.8675,E1 25.0569,E2 381.0746} C_DIS
LIN {X 41.8581,Y 103.2943,Z 112,A 63.3254,B 24.9315,C -1.9112,E1 25.0605,E2 382.446} C_DIS
LIN {X 45.7066,Y 101.6499,Z 112,A 60.7799,B 24.9329,C -1.892,E1 25.0671,E2 385.0307} C_DIS
LIN {X 49.3921,Y 99.911,Z 112,A 58.7698,B 24.9329,C -1.8931,E1 25.0721,E2 387.033} C_DIS
LIN {X 52.657,Y 98.231,Z 112,A 56.8073,B 24.9332,C -1.8873,E1 25.077,E2 389.0036} C_DIS
LIN {X 56.0648,Y 96.327,Z 112,A 54.7047,B 24.9337,C -1.8803,E1 25.0821,E2 391.1165} C_DIS
LIN {X 59.7332,Y 94.0959,Z 112,A 52.5098,B 24.9339,C -1.8775,E1 25.0873,E2 393.3112} C_DIS
LIN {X 63.1073,Y 91.8673,Z 112,A 50.4886,B 24.9339,C -1.8765,E1 25.092,E2 395.3279} C_DIS
LIN {X 66.109,Y 89.7301,Z 112,A 48.7851,B 24.9336,C -1.8815,E1 25.0958,E2 397.0135} C_DIS
LIN {X 69.0951,Y 87.4508,Z 112,A 46.8553,B 24.9339,C -1.878,E1 25.1001,E2 398.9444} C_DIS
LIN {X 71.7526,Y 85.2866,Z 112,A 44.991,B 24.9344,C -1.8702,E1 25.1041,E2 400.8202} C_DIS
LIN {X 74.4393,Y 82.9493,Z 112,A 43.2583,B 24.9344,C -1.8708,E1 25.1077,E2 402.5445} C_DIS
LIN {X 77.0803,Y 80.5019,Z 112,A 41.3594,B 24.9348,C -1.8649,E1 25.1116,E2 404.4496} C_DIS
LIN {X 79.4636,Y 78.1497,Z 112,A 39.6644,B 24.935,C -1.8623,E1 25.1149,E2 406.1435} C_DIS
LIN {X 82.6074,Y 74.8213,Z 112,A 37.2069,B 24.9357,C -1.8525,E1 25.1196,E2 408.6134} C_DIS
LIN {X 84.7576,Y 72.3737,Z 112,A 35.6548,B 24.9356,C -1.854,E1 25.1224,E2 410.1549} C_DIS
LIN {X 87.2816,Y 69.3092,Z 112,A 33.6478,B 24.9358,C -1.8506,E1 25.126,E2 412.1606} C_DIS
LIN {X 89.533,Y 66.3781,Z 112,A 31.6045,B 24.9366,C -1.8396,E1 25.1294,E2 414.2202} C_DIS
LIN {X 91.6821,Y 63.3739,Z 112,A 29.9076,B 24.9363,C -1.8437,E1 25.1321,E2 415.8991} C_DIS
LIN {X 93.7266,Y 60.3086,Z 112,A 27.9917,B 24.9367,C -1.8378,E1 25.1351,E2 417.8193} C_DIS
LIN {X 95.4778,Y 57.4976,Z 112,A 26.1268,B 24.9375,C -1.8261,E1 25.1378,E2 419.7024} C_DIS
LIN {X 97.3237,Y 54.3128,Z 112,A 24.3958,B 24.9374,C -1.8281,E1 25.1402,E2 421.4196} C_DIS
LIN {X 99.0751,Y 51.0493,Z 112,A 22.4608,B 24.9378,C -1.8215,E1 25.1427,E2 423.3602} C_DIS
LIN {X 100.7283,Y 47.7071,Z 112,A 20.5366,B 24.9382,C -1.8157,E1 25.145,E2 425.2876} C_DIS
LIN {X 101.8994,Y 45.1525,Z 112,A 19.0199,B 24.9387,C -1.8083,E1 25.1468,E2 426.8135} C_DIS
LIN {X 103.2566,Y 41.9507,Z 112,A 17.3932,B 24.9386,C -1.8103,E1 25.1485,E2 428.4265} C_DIS
LIN {X 105.1686,Y 36.8965,Z 112,A 14.6583,B 24.939,C -1.804,E1 25.1512,E2 431.1611} C_DIS
LIN {X 106.2132,Y 33.7764,Z 112,A 12.465,B 24.9409,C -1.7764,E1 25.1531,E2 433.407} C_DIS
LIN {X 107.2725,Y 30.2392,Z 112,A 11.111,B 24.9396,C -1.7949,E1 25.1541,E2 434.7095} C_DIS
LIN {X 108.189,Y 26.778,Z 112,A 9.1878,B 24.9402,C -1.7855,E1 25.1554,E2 436.6438} C_DIS
LIN {X 108.9904,Y 23.3043,Z 112,A 7.4215,B 24.9404,C -1.7828,E1 25.1565,E2 438.4063} C_DIS
LIN {X 109.6615,Y 19.9039,Z 112,A 5.5927,B 24.9409,C -1.7751,E1 25.1575,E2 440.2426} C_DIS
LIN {X 110.3027,Y 15.9745,Z 112,A 3.5816,B 24.9413,C -1.7702,E1 25.1583,E2 442.2534} C_DIS
LIN {X 110.7743,Y 12.2997,Z 112,A 1.6933,B 24.9416,C -1.7648,E1 25.1589,E2 444.1432} C_DIS
LIN {X 111.0997,Y 8.8683,Z 112,A 0.0204,B 24.9417,C -1.7636,E1 25.1594,E2 445.809} C_DIS
LIN {X 111.3134,Y 5.6045,Z 112,A -1.7547,B 24.9423,C -1.7539,E1 25.1596,E2 447.5964} C_DIS
LIN {X 111.4368,Y 1.9093,Z 112,A -3.6243,B 24.9427,C -1.7492,E1 25.1598,E2 449.4661} C_DIS
LIN {X 111.4325,Y -2.1431,Z 112,A -5.5889,B 24.9427,C -1.7478,E1 25.1598,E2 451.4223} C_DIS
LIN {X 111.3434,Y -4.9445,Z 112,A -7.0867,B 24.9432,C -1.7405,E1 25.1596,E2 452.9283} C_DIS
LIN {X 111.1193,Y -8.6231,Z 112,A -9.0351,B 24.9438,C -1.7319,E1 25.1592,E2 454.8854} C_DIS
LIN {X 110.7847,Y -12.202,Z 112,A -10.8946,B 24.9442,C -1.7254,E1 25.1587,E2 456.7493} C_DIS
LIN {X 110.2942,Y -16.034,Z 112,A -12.9411,B 24.9448,C -1.7162,E1 25.1579,E2 458.8054} C_DIS
LIN {X 109.745,Y -19.4398,Z 112,A -14.549,B 24.9447,C -1.7179,E1 25.1571,E2 460.3998} C_DIS
LIN {X 109.1202,Y -22.6854,Z 112,A -16.1548,B 24.9447,C -1.7167,E1 25.1563,E2 461.9992} C_DIS
LIN {X 108.4121,Y -25.8636,Z 112,A -17.9266,B 24.9454,C -1.7068,E1 25.1551,E2 463.7839} C_DIS
LIN {X 107.5906,Y -29.087,Z 112,A -19.5838,B 24.9456,C -1.7038,E1 25.154,E2 465.4387} C_DIS
LIN {X 106.3294,Y -33.4068,Z 112,A -21.7167,B 24.9456,C -1.7046,E1 25.1523,E2 467.5575} C_DIS
LIN {X 103.9947,Y -40.0913,Z 112,A -25.4142,B 24.9464,C -1.6905,E1 25.1488,E2 471.2675} C_DIS
LIN {X 102.507,Y -43.7534,Z 112,A -27.5451,B 24.9471,C -1.6798,E1 25.1465,E2 473.412} C_DIS
LIN {X 100.7502,Y -47.6616,Z 112,A -29.8504,B 24.9478,C -1.6684,E1 25.1438,E2 475.7315} C_DIS
LIN {X 99.1613,Y -50.8807,Z 112,A -32.0713,B 24.9492,C -1.6461,E1 25.141,E2 477.9933} C_DIS
LIN {X 97.3083,Y -54.3404,Z 112,A -33.4828,B 24.9479,C -1.6673,E1 25.1391,E2 479.3474} C_DIS
LIN {X 95.6479,Y -57.2154,Z 112,A -35.4884,B 24.9491,C -1.6489,E1 25.1362,E2 481.3861} C_DIS
LIN {X 92.3602,Y -62.381,Z 112,A -38.406,B 24.949,C -1.6503,E1 25.1318,E2 484.2858} C_DIS
LIN {X 90.394,Y -65.2,Z 112,A -40.2631,B 24.9495,C -1.6413,E1 25.1288,E2 486.1551} C_DIS
LIN {X 87.8773,Y -68.5546,Z 112,A -42.2917,B 24.9495,C -1.6411,E1 25.1254,E2 488.1745} C_DIS
LIN {X 85.6134,Y -71.3594,Z 112,A -44.0626,B 24.9496,C -1.6399,E1 25.1223,E2 489.9401} C_DIS
LIN {X 83.4151,Y -73.919,Z 112,A -45.8879,B 24.9501,C -1.6313,E1 25.1189,E2 491.7774} C_DIS
LIN {X 81.1277,Y -76.4205,Z 112,A -47.5626,B 24.9502,C -1.63,E1 25.1157,E2 493.448} C_DIS
LIN {X 78.7368,Y -78.8837,Z 112,A -49.4594,B 24.9508,C -1.6197,E1 25.112,E2 495.3609} C_DIS
LIN {X 76.4343,Y -81.1147,Z 112,A -50.9703,B 24.9508,C -1.6219,E1 25.1089,E2 496.8605} C_DIS
LIN {X 73.9244,Y -83.4102,Z 112,A -52.7238,B 24.951,C -1.6175,E1 25.1053,E2 498.6172} C_DIS
LIN {X 71.3375,Y -85.6315,Z 112,A -54.4666,B 24.9512,C -1.614,E1 25.1016,E2 500.3616} C_DIS
LIN {X 68.7901,Y -87.6919,Z 112,A -56.0533,B 24.9512,C -1.6146,E1 25.0981,E2 501.9409} C_DIS
LIN {X 66.9168,Y -89.1287,Z 112,A -57.3144,B 24.9514,C -1.6099,E1 25.0953,E2 503.2085} C_DIS
LIN {X 63.9017,Y -91.3153,Z 112,A -59.24,B 24.9517,C -1.6054,E1 25.0909,E2 505.138} C_DIS
LIN {X 61.2697,Y -93.1011,Z 112,A -60.8506,B 24.9518,C -1.6033,E1 25.0872,E2 506.7483} C_DIS
LIN {X 58.1464,Y -95.0835,Z 112,A -62.9505,B 24.9526,C -1.5909,E1 25.0822,E2 508.8706} C_DIS
LIN {X 54.5288,Y -97.2031,Z 112,A -64.9098,B 24.9523,C -1.5956,E1 25.0774,E2 510.8131} C_DIS
LIN {X 51.3948,Y -98.8976,Z 112,A -67.3431,B 24.954,C -1.5662,E1 25.0713,E2 513.3089} C_DIS
LIN {X 47.5806,Y -100.7881,Z 112,A -68.8128,B 24.9524,C -1.5939,E1 25.0678,E2 514.7093} C_DIS
LIN {X 44.9663,Y -101.9805,Z 112,A -70.4298,B 24.9529,C -1.5856,E1 25.0636,E2 516.3421} C_DIS
LIN {X 41.7887,Y -103.3225,Z 112,A -72.1346,B 24.9529,C -1.586,E1 25.0592,E2 518.042} C_DIS
LIN {X 35.6015,Y -105.614,Z 112,A -75.1501,B 24.9522,C -1.5978,E1 25.0514,E2 521.0231} C_DIS
LIN {X 33.223,Y -106.3864,Z 112,A -76.8379,B 24.9533,C -1.5788,E1 25.0468,E2 522.7529} C_DIS
LIN {X 30.1311,Y -107.3031,Z 112,A -78.4437,B 24.9533,C -1.5792,E1 25.0425,E2 524.355} C_DIS
LIN {X 24.9635,Y -108.6215,Z 112,A -81.1456,B 24.9533,C -1.5781,E1 25.0352,E2 527.0555} C_DIS
LIN {X 22.5532,Y -109.1474,Z 112,A -82.4871,B 24.9536,C -1.5738,E1 25.0315,E2 528.4053} C_DIS
LIN {X 19.221,Y -109.7843,Z 112,A -84.2387,B 24.9536,C -1.572,E1 25.0267,E2 530.1592} C_DIS
LIN {X 15.8153,Y -110.3253,Z 112,A -86.0043,B 24.9538,C -1.5711,E1 25.0218,E2 531.9253} C_DIS
LIN {X 12.2699,Y -110.7776,Z 112,A -87.875,B 24.9539,C -1.5685,E1 25.0166,E2 533.8008} C_DIS
LIN {X 8.6326,Y -111.1185,Z 112,A -89.6724,B 24.9538,C -1.571,E1 25.0116,E2 535.5913} C_DIS
LIN {X 5.0086,Y -111.3407,Z 112,A -91.6297,B 24.954,C -1.5664,E1 25.0061,E2 537.5588} C_DIS
LIN {X 0.7849,Y -111.4486,Z 112,A -93.661,B 24.9537,C -1.5718,E1 25.0005,E2 539.5771} C_DIS
Enddeposition()
LIN {X 0.7849,Y -111.4486,Z 112,A -93.661,B 24.9537,C -1.5718,E1 25.0005,E2 539.5771} C_DIS
Startdeposition()
$VEL.CP = VEL_PRINT
LIN {X 1.8726,Y -110.5064,Z 112,A -92.4883,B 24.9512,C -1.6139,E1 25.004,E2 538.3045} C_DIS
LIN {X 4.8709,Y -110.4149,Z 112,A -90.8254,B 24.9509,C -1.6191,E1 25.0087,E2 536.6299} C_DIS
LIN {X 8.7451,Y -110.1757,Z 112,A -88.8831,B 24.951,C -1.617,E1 25.0141,E2 534.6934} C_DIS
LIN {X 12.1524,Y -109.8539,Z 112,A -87.0051,B 24.9507,C -1.6224,E1 25.0194,E2 532.8038} C_DIS
LIN {X 15.6399,Y -109.41,Z 112,A -85.2212,B 24.9507,C -1.622,E1 25.0243,E2 531.0224} C_DIS
LIN {X 19.446,Y -108.7981,Z 112,A -83.2581,B 24.9507,C -1.622,E1 25.0297,E2 529.0613} C_DIS
LIN {X 23.2272,Y -108.0544,Z 112,A -80.9933,B 24.9499,C -1.6354,E1 25.036,E2 526.7678} C_DIS
LIN {X 28.2221,Y -106.86,Z 112,A -78.094,B 24.9491,C -1.6484,E1 25.0439,E2 523.842} C_DIS
LIN {X 31.9638,Y -105.8006,Z 112,A -76.5354,B 24.9502,C -1.6307,E1 25.0479,E2 522.328} C_DIS
LIN {X 35.2544,Y -104.7487,Z 112,A -73.9571,B 24.9479,C -1.6676,E1 25.055,E2 519.6675} C_DIS
LIN {X 40.2953,Y -102.9148,Z 112,A -72.0539,B 24.95,C -1.6328,E1 25.0597,E2 517.8508} C_DIS
LIN {X 43.6071,Y -101.5576,Z 112,A -70.3064,B 24.9502,C -1.6307,E1 25.0642,E2 516.1122} C_DIS
LIN {X 47.0377,Y -100.014,Z 112,A -68.421,B 24.9502,C -1.6309,E1 25.069,E2 514.2311} C_DIS
LIN {X 53.9643,Y -96.4522,Z 112,A -64.2216,B 24.9493,C -1.6448,E1 25.0794,E2 510.0106} C_DIS
LIN {X 58.518,Y -93.7593,Z 112,A -61.3568,B 24.9487,C -1.6554,E1 25.0863,E2 507.1298} C_DIS
LIN {X 61.8258,Y -91.612,Z 112,A -59.497,B 24.9489,C -1.6512,E1 25.0906,E2 505.2859} C_DIS
LIN {X 64.274,Y -89.9112,Z 112,A -57.9272,B 24.9486,C -1.6555,E1 25.0942,E2 503.7114} C_DIS
LIN {X 66.3839,Y -88.3648,Z 112,A -56.3628,B 24.9479,C -1.6677,E1 25.0977,E2 502.124} C_DIS
LIN {X 70.3166,Y -85.2696,Z 112,A -53.9323,B 24.9479,C -1.6661,E1 25.103,E2 499.7064} C_DIS
LIN {X 73.0614,Y -82.9302,Z 112,A -52.1001,B 24.9479,C -1.6687,E1 25.1068,E2 497.8752} C_DIS
LIN {X 76.0285,Y -80.2185,Z 112,A -49.9505,B 24.9473,C -1.6766,E1 25.1113,E2 495.7157} C_DIS
LIN {X 78.9898,Y -77.3048,Z 112,A -47.8692,B 24.9472,C -1.6786,E1 25.1154,E2 493.6384} C_DIS
LIN {X 81.4597,Y -74.6958,Z 112,A -46.0713,B 24.9471,C -1.6805,E1 25.1188,E2 491.844} C_DIS
LIN {X 83.7987,Y -72.0638,Z 112,A -44.107,B 24.9464,C -1.6914,E1 25.1224,E2 489.8627} C_DIS
LIN {X 87.0849,Y -68.0568,Z 112,A -41.487,B 24.9461,C -1.6956,E1 25.127,E2 487.2451} C_DIS
LIN {X 89.2943,Y -65.1285,Z 112,A -39.7123,B 24.9461,C -1.6951,E1 25.1299,E2 485.48} C_DIS
LIN {X 92.4327,Y -60.5924,Z 112,A -36.8992,B 24.9458,C -1.701,E1 25.1343,E2 482.6668} C_DIS
LIN {X 94.7414,Y -56.9148,Z 112,A -34.4288,B 24.9447,C -1.7175,E1 25.138,E2 480.1703} C_DIS
LIN {X 96.8993,Y -53.1578,Z 112,A -31.8757,B 24.9434,C -1.738,E1 25.1415,E2 477.582} C_DIS
LIN {X 98.7195,Y -49.6998,Z 112,A -30.3267,B 24.9444,C -1.7224,E1 25.1434,E2 476.0781} C_DIS
LIN {X 101.0677,Y -44.7309,Z 112,A -27.4388,B 24.9437,C -1.7328,E1 25.1468,E2 473.1813} C_DIS
LIN {X 102.5097,Y -41.3164,Z 112,A -25.7506,B 24.944,C -1.7282,E1 25.1486,E2 471.5133} C_DIS
LIN {X 104.0972,Y -37.1384,Z 112,A -23.1231,B 24.9426,C -1.7495,E1 25.1512,E2 468.8502} C_DIS
LIN {X 105.4459,Y -33.1131,Z 112,A -21.2083,B 24.943,C -1.7434,E1 25.1528,E2 466.9605} C_DIS
LIN {X 106.1126,Y -30.912,Z 112,A -20.0119,B 24.9428,C -1.7474,E1 25.1537,E2 465.7616} C_DIS
LIN {X 106.93,Y -27.9524,Z 112,A -18.3402,B 24.9422,C -1.7561,E1 25.155,E2 464.0789} C_DIS
LIN {X 107.7231,Y -24.7166,Z 112,A -16.6068,B 24.9418,C -1.762,E1 25.1561,E2 462.3418} C_DIS
LIN {X 108.4835,Y -21.1312,Z 112,A -14.7614,B 24.9416,C -1.7656,E1 25.1571,E2 460.4986} C_DIS
LIN {X 109.4189,Y -15.5776,Z 112,A -11.9044,B 24.9411,C -1.7722,E1 25.1584,E2 457.6428} C_DIS
LIN {X 109.8428,Y -12.2508,Z 112,A -10.0382,B 24.9404,C -1.7836,E1 25.159,E2 455.7607} C_DIS
LIN {X 110.1794,Y -8.6986,Z 112,A -8.314,B 24.9404,C -1.784,E1 25.1594,E2 454.0459} C_DIS
LIN {X 110.4133,Y -4.9073,Z 112,A -6.4284,B 24.9402,C -1.7866,E1 25.1597,E2 452.1653} C_DIS
LIN {X 110.5049,Y -1.9553,Z 112,A -4.8362,B 24.9397,C -1.7943,E1 25.1597,E2 450.5644} C_DIS
LIN {X 110.5055,Y 1.9236,Z 112,A -2.8599,B 24.9393,C -1.7993,E1 25.1597,E2 448.5881} C_DIS
LIN {X 110.3907,Y 5.4306,Z 112,A -0.9314,B 24.9386,C -1.8101,E1 25.1595,E2 446.6456} C_DIS
LIN {X 110.1747,Y 8.7567,Z 112,A 0.6489,B 24.9386,C -1.809,E1 25.1592,E2 445.0772} C_DIS
LIN {X 109.8473,Y 12.212,Z 112,A 2.5495,B 24.938,C -1.8193,E1 25.1586,E2 443.1636} C_DIS
LIN {X 109.3989,Y 15.7185,Z 112,A 4.2866,B 24.9379,C -1.8209,E1 25.158,E2 441.433} C_DIS
LIN {X 108.8002,Y 19.4342,Z 112,A 6.267,B 24.9373,C -1.8284,E1 25.1571,E2 439.4466} C_DIS
LIN {X 108.0791,Y 23.114,Z 112,A 8.18,B 24.937,C -1.8331,E1 25.156,E2 437.5337} C_DIS
LIN {X 107.3334,Y 26.3576,Z 112,A 10.0993,B 24.936,C -1.8472,E1 25.1547,E2 435.5921} C_DIS
LIN {X 106.413,Y 29.858,Z 112,A 12.4125,B 24.9343,C -1.8728,E1 25.153,E2 433.2318} C_DIS
LIN {X 105.1037,Y 34.1818,Z 112,A 14.0434,B 24.936,C -1.8477,E1 25.1516,E2 431.6695} C_DIS
LIN {X 104.2329,Y 36.7515,Z 112,A 15.8689,B 24.9344,C -1.8708,E1 25.1499,E2 429.7996} C_DIS
LIN {X 103.0402,Y 39.9761,Z 112,A 17.2834,B 24.9352,C -1.8594,E1 25.1485,E2 428.4198} C_DIS
LIN {X 101.7719,Y 43.1007,Z 112,A 18.9749,B 24.935,C -1.862,E1 25.1467,E2 426.7316} C_DIS
LIN {X 100.5308,Y 45.9242,Z 112,A 21.113,B 24.933,C -1.8908,E1 25.1442,E2 424.537} C_DIS
LIN {X 98.8086,Y 49.5202,Z 112,A 22.6765,B 24.9342,C -1.874,E1 25.1423,E2 423.0217} C_DIS
LIN {X 96.8648,Y 53.2233,Z 112,A 25.3954,B 24.932,C -1.9047,E1 25.1386,E2 420.2445} C_DIS
LIN {X 94.7215,Y 56.9497,Z 112,A 27.0189,B 24.9335,C -1.8835,E1 25.1363,E2 418.6793} C_DIS
LIN {X 93.1054,Y 59.5531,Z 112,A 28.4801,B 24.9335,C -1.8821,E1 25.1342,E2 417.229} C_DIS
LIN {X 91.1315,Y 62.5348,Z 112,A 30.5082,B 24.9327,C -1.8946,E1 25.131,E2 415.1814} C_DIS
LIN {X 89.0012,Y 65.5288,Z 112,A 32.4216,B 24.9323,C -1.8997,E1 25.1278,E2 413.265} C_DIS
LIN {X 87.265,Y 67.8247,Z 112,A 34.1828,B 24.9312,C -1.9153,E1 25.1248,E2 411.4753} C_DIS
LIN {X 85.203,Y 70.3967,Z 112,A 35.5048,B 24.9322,C -1.9022,E1 25.1225,E2 410.1905} C_DIS
LIN {X 83.252,Y 72.6929,Z 112,A 37.0279,B 24.932,C -1.9041,E1 25.1197,E2 408.6697} C_DIS
LIN {X 80.8121,Y 75.3972,Z 112,A 38.984,B 24.9315,C -1.9113,E1 25.116,E2 406.7052} C_DIS
LIN {X 78.4977,Y 77.8029,Z 112,A 40.7081,B 24.9313,C -1.9148,E1 25.1126,E2 404.9802} C_DIS
LIN {X 75.6871,Y 80.5395,Z 112,A 42.6737,B 24.9312,C -1.9161,E1 25.1087,E2 403.0197} C_DIS
LIN {X 73.0199,Y 82.9664,Z 112,A 44.5728,B 24.9308,C -1.9212,E1 25.1047,E2 401.1162} C_DIS
LIN {X 70.5783,Y 85.0521,Z 112,A 46.2224,B 24.9306,C -1.9237,E1 25.1012,E2 399.467} C_DIS
LIN {X 68.5203,Y 86.7186,Z 112,A 47.7875,B 24.9298,C -1.9347,E1 25.0977,E2 397.8818} C_DIS
LIN {X 64.974,Y 89.4074,Z 112,A 49.8669,B 24.9303,C -1.9288,E1 25.0931,E2 395.8237} C_DIS
LIN {X 62.3225,Y 91.2756,Z 112,A 51.9871,B 24.9287,C -1.9508,E1 25.0881,E2 393.6588} C_DIS
LIN {X 59.3143,Y 93.2587,Z 112,A 53.4941,B 24.9296,C -1.938,E1 25.0847,E2 392.187} C_DIS
LIN {X 56.4845,Y 94.9986,Z 112,A 55.6862,B 24.9279,C -1.961,E1 25.0793,E2 389.9473} C_DIS
LIN {X 52.9175,Y 97.0307,Z 112,A 57.2238,B 24.9296,C -1.9383,E1 25.0757,E2 388.4677} C_DIS
LIN {X 50.095,Y 98.5175,Z 112,A 58.8425,B 24.9296,C -1.939,E1 25.0717,E2 386.8518} C_DIS
LIN {X 45.4507,Y 100.7442,Z 112,A 61.5131,B 24.9293,C -1.9422,E1 25.0649,E2 384.1806} C_DIS
LIN {X 42.4204,Y 102.0586,Z 112,A 63.3236,B 24.9288,C -1.9482,E1 25.0602,E2 382.36} C_DIS
LIN {X 35.7803,Y 104.5703,Z 112,A 67.0765,B 24.9284,C -1.9547,E1 25.0504,E2 378.5996} C_DIS
LIN {X 32.4442,Y 105.6533,Z 112,A 69.0251,B 24.9279,C -1.9617,E1 25.0452,E2 376.6381} C_DIS
LIN {X 27.7339,Y 106.9861,Z 112,A 71.3576,B 24.9284,C -1.9546,E1 25.0389,E2 374.326} C_DIS
LIN {X 23.8806,Y 107.9119,Z 112,A 73.2665,B 24.9287,C -1.9496,E1 25.0338,E2 372.4317} C_DIS
LIN {X 21.1764,Y 108.4749,Z 112,A 74.688,B 24.9287,C -1.9498,E1 25.0299,E2 371.0115} C_DIS
LIN {X 17.6162,Y 109.111,Z 112,A 76.6991,B 24.9283,C -1.9562,E1 25.0243,E2 368.9874} C_DIS
LIN {X 14.3594,Y 109.5855,Z 112,A 78.3527,B 24.9283,C -1.9544,E1 25.0198,E2 367.3393} C_DIS
LIN {X 10.6595,Y 110.0081,Z 112,A 80.3108,B 24.9283,C -1.9558,E1 25.0143,E2 365.3792} C_DIS
LIN {X 7.684,Y 110.255,Z 112,A 81.7358,B 24.9286,C -1.9508,E1 25.0104,E2 363.9668} C_DIS
LIN {X 4.4833,Y 110.4315,Z 112,A 83.5337,B 24.9282,C -1.9564,E1 25.0053,E2 362.1562} C_DIS
LIN {X 0.8267,Y 110.5192,Z 112,A 85.3801,B 24.9284,C -1.9541,E1 25.0002,E2 360.3156} C_DIS
LIN {X -2.789,Y 110.4886,Z 112,A 87.3186,B 24.9283,C -1.9562,E1 24.9948,E2 358.372} C_DIS
LIN {X -6.1813,Y 110.3492,Z 112,A 89.0185,B 24.9285,C -1.9531,E1 24.99,E2 356.6789} C_DIS
LIN {X -10.0211,Y 110.067,Z 112,A 91.0192,B 24.9285,C -1.9524,E1 24.9845,E2 354.679} C_DIS
LIN {X -13.6607,Y 109.676,Z 112,A 92.9789,B 24.9285,C -1.9538,E1 24.979,E2 352.7147} C_DIS
LIN {X -16.6483,Y 109.2614,Z 112,A 95.1247,B 24.9267,C -1.9767,E1 24.973,E2 350.5127} C_DIS
LIN {X -20.9804,Y 108.5126,Z 112,A 96.7531,B 24.9288,C -1.9482,E1 24.9687,E2 348.9501} C_DIS
LIN {X -24.6496,Y 107.7386,Z 112,A 98.6983,B 24.929,C -1.9466,E1 24.9634,E2 347.0065} C_DIS
LIN {X -27.7536,Y 106.9811,Z 112,A 100.4628,B 24.9288,C -1.9493,E1 24.9586,E2 345.2329} C_DIS
LIN {X -34.6694,Y 104.9459,Z 112,A 104.2057,B 24.9291,C -1.9452,E1 24.9486,E2 341.4933} C_DIS
LIN {X -37.9867,Y 103.7891,Z 112,A 106.1412,B 24.9289,C -1.9475,E1 24.9435,E2 339.5485} C_DIS
LIN {X -41.8374,Y 102.2977,Z 112,A 108.1106,B 24.9296,C -1.9377,E1 24.9384,E2 337.5981} C_DIS
LIN {X -45.6556,Y 100.6518,Z 112,A 111.2024,B 24.9271,C -1.9722,E1 24.9303,E2 334.4169} C_DIS
LIN {X -50.8132,Y 98.1504,Z 112,A 113.0906,B 24.9306,C -1.9238,E1 24.9259,E2 332.6387} C_DIS
LIN {X -55.0989,Y 95.8085,Z 112,A 115.7986,B 24.9304,C -1.9263,E1 24.9192,E2 329.9168} C_DIS
LIN {X -58.749,Y 93.615,Z 112,A 118.3384,B 24.9298,C -1.9354,E1 24.9131,E2 327.3475} C_DIS
LIN {X -61.4596,Y 91.8599,Z 112,A 120.3935,B 24.9289,C -1.9473,E1 24.9083,E2 325.2573} C_DIS
LIN {X -65.2502,Y 89.2052,Z 112,A 122.0283,B 24.9315,C -1.9121,E1 24.9048,E2 323.7006} C_DIS
LIN {X -68.6411,Y 86.6231,Z 112,A 124.3124,B 24.9315,C -1.9103,E1 24.8997,E2 321.4124} C_DIS
LIN {X -70.7125,Y 84.9406,Z 112,A 126.0546,B 24.9308,C -1.9213,E1 24.8959,E2 319.6373} C_DIS
LIN {X -73.2318,Y 82.7809,Z 112,A 127.535,B 24.9318,C -1.9079,E1 24.8928,E2 318.183} C_DIS
LIN {X -75.3635,Y 80.8439,Z 112,A 129.5851,B 24.9304,C -1.9263,E1 24.8886,E2 316.0807} C_DIS
LIN {X -78.5295,Y 77.7707,Z 112,A 131.1823,B 24.9328,C -1.8936,E1 24.8855,E2 314.5545} C_DIS
LIN {X -82.1021,Y 73.99,Z 112,A 133.971,B 24.933,C -1.8904,E1 24.8802,E2 311.7612} C_DIS
LIN {X -85.6862,Y 69.8076,Z 112,A 136.8783,B 24.9334,C -1.885,E1 24.875,E2 308.8535} C_DIS
LIN {X -89.7703,Y 64.4714,Z 112,A 140.3263,B 24.9342,C -1.8741,E1 24.8692,E2 305.4149} C_DIS
LIN {X -91.6285,Y 61.8013,Z 112,A 142.3415,B 24.9336,C -1.8822,E1 24.866,E2 303.3705} C_DIS
LIN {X -93.3827,Y 59.1208,Z 112,A 143.7426,B 24.9346,C -1.8674,E1 24.864,E2 301.9976} C_DIS
LIN {X -94.836,Y 56.7596,Z 112,A 145.4344,B 24.9342,C -1.8731,E1 24.8615,E2 300.2835} C_DIS
LIN {X -96.9895,Y 52.9935,Z 112,A 147.4846,B 24.9352,C -1.8588,E1 24.8587,E2 298.2565} C_DIS
LIN {X -98.9065,Y 49.3226,Z 112,A 150.2939,B 24.9339,C -1.8781,E1 24.8552,E2 295.3861} C_DIS
LIN {X -100.9745,Y 44.9395,Z 112,A 152.1737,B 24.9361,C -1.8459,E1 24.8531,E2 293.5727} C_DIS
LIN {X -102.3912,Y 41.6076,Z 112,A 154.8946,B 24.9342,C -1.8729,E1 24.8501,E2 290.7724} C_DIS
LIN {X -104.3612,Y 36.3859,Z 112,A 156.9507,B 24.9371,C -1.8314,E1 24.8483,E2 288.8036} C_DIS
LIN {X -105.5015,Y 32.9338,Z 112,A 158.9871,B 24.9371,C -1.8313,E1 24.8465,E2 286.7558} C_DIS
LIN {X -107.3391,Y 26.3341,Z 112,A 162.5034,B 24.938,C -1.8186,E1 24.844,E2 283.2492} C_DIS
LIN {X -108.1057,Y 22.992,Z 112,A 164.0428,B 24.939,C -1.8037,E1 24.8431,E2 281.7362} C_DIS
LIN {X -108.7579,Y 19.6694,Z 112,A 165.9703,B 24.939,C -1.8047,E1 24.8421,E2 279.7951} C_DIS
LIN {X -109.4076,Y 15.657,Z 112,A 167.997,B 24.9396,C -1.7948,E1 24.8412,E2 277.7799} C_DIS
LIN {X -109.8327,Y 12.3372,Z 112,A 169.8603,B 24.9396,C -1.7941,E1 24.8406,E2 275.9072} C_DIS
LIN {X -110.2902,Y 7.1636,Z 112,A 172.3828,B 24.9407,C -1.7788,E1 24.8401,E2 273.4059} C_DIS
LIN {X -110.4937,Y 2.5636,Z 112,A 174.9391,B 24.9407,C -1.7775,E1 24.8398,E2 270.8373} C_DIS
LIN {X -110.5215,Y -0.5642,Z 112,A 176.3758,B 24.9416,C -1.7652,E1 24.8398,E2 269.4213} C_DIS
LIN {X -110.4402,Y -4.2803,Z 112,A 178.6495,B 24.9411,C -1.7723,E1 24.84,E2 267.117} C_DIS
LIN {X -110.1797,Y -8.6942,Z 112,A -179.2654,B 24.9421,C -1.757,E1 24.8404,E2 265.0559} C_DIS
LIN {X -109.8745,Y -11.9558,Z 112,A -177.671,B 24.9428,C -1.7475,E1 24.8408,E2 263.4745} C_DIS
LIN {X -109.4461,Y -15.3862,Z 112,A -175.2868,B 24.9416,C -1.7646,E1 24.8417,E2 261.0352} C_DIS
LIN {X -108.8997,Y -18.8782,Z 112,A -173.744,B 24.9428,C -1.7476,E1 24.8424,E2 259.5238} C_DIS
LIN {X -108.1389,Y -22.8368,Z 112,A -171.4862,B 24.9428,C -1.7476,E1 24.8437,E2 257.2528} C_DIS
LIN {X -106.9309,Y -27.9489,Z 112,A -168.8222,B 24.9435,C -1.7369,E1 24.8455,E2 254.5988} C_DIS
LIN {X -105.7584,Y -32.1052,Z 112,A -166.6871,B 24.9442,C -1.726,E1 24.8472,E2 252.4772} C_DIS
LIN {X -104.7186,Y -35.3437,Z 112,A -164.9657,B 24.9446,C -1.7191,E1 24.8487,E2 250.7624} C_DIS
LIN {X -103.3842,Y -39.0751,Z 112,A -162.9293,B 24.9451,C -1.7123,E1 24.8506,E2 248.7308} C_DIS
LIN {X -101.5695,Y -43.5799,Z 112,A -160.4765,B 24.9457,C -1.7024,E1 24.8532,E2 246.2878} C_DIS
LIN {X -99.8955,Y -47.2899,Z 112,A -158.0833,B 24.9454,C -1.7075,E1 24.856,E2 243.8696} C_DIS
LIN {X -97.97,Y -51.1585,Z 112,A -155.9797,B 24.9461,C -1.6959,E1 24.8587,E2 241.7823} C_DIS
LIN {X -96.4159,Y -54.0292,Z 112,A -154.3159,B 24.9465,C -1.6902,E1 24.8609,E2 240.1234} C_DIS
LIN {X -94.3279,Y -57.5973,Z 112,A -150.9316,B 24.9437,C -1.7336,E1 24.8661,E2 236.6182} C_DIS
LIN {X -90.6019,Y -63.2971,Z 112,A -148.8919,B 24.948,C -1.6655,E1 24.869,E2 234.7307} C_DIS
LIN {X -87.6219,Y -67.3615,Z 112,A -145.9558,B 24.9476,C -1.6717,E1 24.8739,E2 231.7657} C_DIS
LIN {X -85.2217,Y -70.3742,Z 112,A -144.0132,B 24.9481,C -1.6648,E1 24.8773,E2 229.8305} C_DIS
LIN {X -83.4445,Y -72.4725,Z 112,A -142.5897,B 24.9483,C -1.6614,E1 24.8799,E2 228.4086} C_DIS
LIN {X -80.3706,Y -75.8668,Z 112,A -140.0854,B 24.9483,C -1.6612,E1 24.8847,E2 225.8935} C_DIS
LIN {X -77.7269,Y -78.5729,Z 112,A -138.1468,B 24.9486,C -1.6561,E1 24.8885,E2 223.9589} C_DIS
LIN {X -74.9898,Y -81.19,Z 112,A -136.1492,B 24.9488,C -1.6535,E1 24.8925,E2 221.9594} C_DIS
LIN {X -72.2724,Y -83.6193,Z 112,A -134.4756,B 24.9495,C -1.6411,E1 24.896,E2 220.3087} C_DIS
LIN {X -68.3993,Y -86.8143,Z 112,A -131.6554,B 24.9493,C -1.6449,E1 24.9022,E2 217.4688} C_DIS
LIN {X -65.8389,Y -88.774,Z 112,A -129.4721,B 24.9482,C -1.6626,E1 24.9072,E2 215.2355} C_DIS
LIN {X -62.6445,Y -91.0555,Z 112,A -127.9052,B 24.9496,C -1.6403,E1 24.9106,E2 213.7165} C_DIS
LIN {X -59.1801,Y -93.3448,Z 112,A -124.8072,B 24.9474,C -1.6755,E1 24.9182,E2 210.5248} C_DIS
LIN {X -54.1412,Y -96.3534,Z 112,A -122.7475,B 24.9502,C -1.6309,E1 24.9229,E2 208.5649} C_DIS
LIN {X -48.4522,Y -99.3376,Z 112,A -119.3371,B 24.9502,C -1.6299,E1 24.9314,E2 205.1478} C_DIS
LIN {X -45.5082,Y -100.7183,Z 112,A -117.7398,B 24.9506,C -1.6244,E1 24.9354,E2 203.5597} C_DIS
LIN {X -42.2593,Y -102.126,Z 112,A -115.4111,B 24.9494,C -1.6427,E1 24.9416,E2 201.182} C_DIS
LIN {X -38.9105,Y -103.4465,Z 112,A -113.9324,B 24.9505,C -1.625,E1 24.9453,E2 199.7424} C_DIS
LIN {X -35.5205,Y -104.6589,Z 112,A -112.0045,B 24.9505,C -1.626,E1 24.9504,E2 197.8085} C_DIS
LIN {X -30.8998,Y -106.1163,Z 112,A -109.4295,B 24.9505,C -1.6268,E1 24.9573,E2 195.2272} C_DIS
LIN {X -26.494,Y -107.3001,Z 112,A -107.2612,B 24.951,C -1.6172,E1 24.9631,E2 193.0785} C_DIS
LIN {X -23.3034,Y -108.0378,Z 112,A -105.5795,B 24.951,C -1.6157,E1 24.9677,E2 191.3982} C_DIS
LIN {X -19.6233,Y -108.7662,Z 112,A -103.6437,B 24.9512,C -1.6146,E1 24.973,E2 189.4629} C_DIS
LIN {X -16.2787,Y -109.3185,Z 112,A -101.7907,B 24.9509,C -1.6181,E1 24.9782,E2 187.5999} C_DIS
LIN {X -12.9625,Y -109.7594,Z 112,A -100.1295,B 24.9511,C -1.6148,E1 24.9827,E2 185.9455} C_DIS
LIN {X -9.5208,Y -110.1132,Z 112,A -98.2205,B 24.9509,C -1.6195,E1 24.9881,E2 184.0244} C_DIS
LIN {X -6.0446,Y -110.3568,Z 112,A -96.4967,B 24.9511,C -1.6161,E1 24.9929,E2 182.308} C_DIS
LIN {X -2.0014,Y -110.5041,Z 112,A -94.3883,B 24.9511,C -1.6168,E1 24.9988,E2 180.1976} C_DIS
LIN {X 0.776,Y -110.5169,Z 112,A -93.2492,B 24.9518,C -1.6045,E1 25.0019,E2 179.0878} C_DIS
Enddeposition()
LIN {X 0.776,Y -110.5169,Z 112,A -93.2492,B 24.9518,C -1.6045,E1 25.0019,E2 179.0878} C_DIS
Startdeposition()
$VEL.CP = VEL_PRINT
LIN {X -0.6877,Y -109.5892,Z 112,A -94.5963,B 24.9523,C -1.5962,E1 24.998,E2 180.4544} C_DIS
LIN {X -4.0265,Y -109.5193,Z 112,A -96.44,B 24.9525,C -1.5919,E1 24.9929,E2 182.3086} C_DIS
LIN {X -7.8209,Y -109.3127,Z 112,A -98.37,B 24.9524,C -1.5942,E1 24.9875,E2 184.2337} C_DIS
LIN {X -11.3412,Y -109.0029,Z 112,A -100.1334,B 24.9522,C -1.5979,E1 24.9826,E2 185.9895} C_DIS
LIN {X -14.672,Y -108.6064,Z 112,A -102.0379,B 24.9525,C -1.592,E1 24.9773,E2 187.9093} C_DIS
LIN {X -18.3844,Y -108.0387,Z 112,A -103.8343,B 24.9521,C -1.5994,E1 24.9724,E2 189.6898} C_DIS
LIN {X -21.3364,Y -107.4961,Z 112,A -105.3688,B 24.952,C -1.6014,E1 24.9682,E2 191.2212} C_DIS
LIN {X -24.3457,Y -106.8534,Z 112,A -107.0984,B 24.9522,C -1.5972,E1 24.9634,E2 192.9628} C_DIS
LIN {X -27.8705,Y -105.9899,Z 112,A -109.2696,B 24.9528,C -1.5873,E1 24.9575,E2 195.1608} C_DIS
LIN {X -33.0897,Y -104.4783,Z 112,A -111.8972,B 24.9522,C -1.5979,E1 24.9505,E2 197.7678} C_DIS
LIN {X -36.1349,Y -103.4628,Z 112,A -113.5062,B 24.9519,C -1.6021,E1 24.9463,E2 199.3698} C_DIS
LIN {X -42.7405,Y -100.9135,Z 112,A -116.9753,B 24.9511,C -1.615,E1 24.9374,E2 202.8158} C_DIS
LIN {X -44.86,Y -99.9893,Z 112,A -118.434,B 24.9517,C -1.6063,E1 24.9336,E2 204.2985} C_DIS
LIN {X -48.0302,Y -98.5076,Z 112,A -120.795,B 24.9528,C -1.5874,E1 24.9275,E2 206.7104} C_DIS
LIN {X -51.5705,Y -96.7009,Z 112,A -122.2471,B 24.9511,C -1.6149,E1 24.9241,E2 208.1013} C_DIS
LIN {X -57.7799,Y -93.1228,Z 112,A -126.0941,B 24.9511,C -1.6163,E1 24.9148,E2 211.9565} C_DIS
LIN {X -60.4423,Y -91.4166,Z 112,A -127.7358,B 24.9509,C -1.6194,E1 24.9109,E2 213.5963} C_DIS
LIN {X -66.4979,Y -87.1122,Z 112,A -132.873,B 24.9534,C -1.5776,E1 24.8991,E2 218.8509} C_DIS
LIN {X -71.7737,Y -82.8189,Z 112,A -135.2963,B 24.9503,C -1.628,E1 24.8942,E2 221.1637} C_DIS
LIN {X -74.5036,Y -80.3727,Z 112,A -137.1925,B 24.9501,C -1.6327,E1 24.8903,E2 223.0565} C_DIS
LIN {X -77.0964,Y -77.8872,Z 112,A -138.986,B 24.9496,C -1.6399,E1 24.8867,E2 224.8403} C_DIS
LIN {X -79.6311,Y -75.2943,Z 112,A -141.5296,B 24.9509,C -1.6191,E1 24.8817,E2 227.4443} C_DIS
LIN {X -82.4343,Y -72.214,Z 112,A -142.7954,B 24.9484,C -1.6591,E1 24.8795,E2 228.6207} C_DIS
LIN {X -85.0953,Y -69.0582,Z 112,A -145.3125,B 24.949,C -1.6503,E1 24.875,E2 231.1703} C_DIS
LIN {X -88.4732,Y -64.6743,Z 112,A -148.1088,B 24.9483,C -1.6611,E1 24.8703,E2 233.9542} C_DIS
LIN {X -90.3348,Y -62.0503,Z 112,A -150.8663,B 24.9505,C -1.6246,E1 24.8658,E2 236.8124} C_DIS
LIN {X -93.4471,Y -57.2542,Z 112,A -152.8979,B 24.9478,C -1.6686,E1 24.8629,E2 238.7494} C_DIS
LIN {X -95.1381,Y -54.3972,Z 112,A -154.6111,B 24.9475,C -1.6741,E1 24.8605,E2 240.4584} C_DIS
LIN {X -96.9992,Y -51.004,Z 112,A -156.5203,B 24.9469,C -1.684,E1 24.858,E2 242.3541} C_DIS
LIN {X -98.4112,Y -48.226,Z 112,A -158.6671,B 24.9478,C -1.669,E1 24.8552,E2 244.5483} C_DIS
LIN {X -100.6301,Y -43.4053,Z 112,A -161.5549,B 24.9476,C -1.6727,E1 24.852,E2 247.4431} C_DIS
LIN {X -101.9626,Y -40.1732,Z 112,A -162.9178,B 24.9461,C -1.6955,E1 24.8506,E2 248.7592} C_DIS
LIN {X -103.0841,Y -37.203,Z 112,A -164.704,B 24.9461,C -1.6957,E1 24.8489,E2 250.5551} C_DIS
LIN {X -104.2746,Y -33.7203,Z 112,A -166.4537,B 24.9453,C -1.7081,E1 24.8473,E2 252.2853} C_DIS
LIN {X -105.0778,Y -31.1273,Z 112,A -167.9947,B 24.9453,C -1.7078,E1 24.8461,E2 253.8358} C_DIS
LIN {X -106.1326,Y -27.3152,Z 112,A -170.8693,B 24.9468,C -1.6841,E1 24.844,E2 256.7837} C_DIS
LIN {X -107.2797,Y -22.393,Z 112,A -172.4952,B 24.9439,C -1.7302,E1 24.8431,E2 258.3092} C_DIS
LIN {X -108.4397,Y -15.8516,Z 112,A -176.7974,B 24.9452,C -1.7102,E1 24.8411,E2 262.6847} C_DIS
LIN {X -108.9529,Y -11.8188,Z 112,A -178.3064,B 24.9433,C -1.7399,E1 24.8406,E2 264.1318} C_DIS
LIN {X -109.2413,Y -8.7519,Z 112,A 179.4454,B 24.9445,C -1.7214,E1 24.8401,E2 266.4378} C_DIS
LIN {X -109.4901,Y -4.7081,Z 112,A 177.2857,B 24.9441,C -1.7267,E1 24.8398,E2 268.5978} C_DIS
LIN {X -109.5911,Y -0.501,Z 112,A 175.6357,B 24.9423,C -1.7542,E1 24.8398,E2 270.1922} C_DIS
LIN {X -109.4105,Y 6.297,Z 112,A 172.3833,B 24.9408,C -1.777,E1 24.8401,E2 273.4097} C_DIS
LIN {X -108.9799,Y 11.5614,Z 112,A 169.4426,B 24.9407,C -1.7792,E1 24.8408,E2 276.3627} C_DIS
LIN {X -108.6787,Y 14.1137,Z 112,A 167.9842,B 24.9407,C -1.7792,E1 24.8413,E2 277.8297} C_DIS
LIN {X -108.0148,Y 18.5278,Z 112,A 165.3508,B 24.9409,C -1.7757,E1 24.8424,E2 280.4875} C_DIS
LIN {X -107.2655,Y 22.4624,Z 112,A 163.4903,B 24.9399,C -1.7911,E1 24.8435,E2 282.3222} C_DIS
LIN {X -106.5074,Y 25.8157,Z 112,A 160.6047,B 24.9422,C -1.7567,E1 24.8455,E2 285.3066} C_DIS
LIN {X -104.8711,Y 31.8238,Z 112,A 158.2959,B 24.9391,C -1.8018,E1 24.8472,E2 287.5212} C_DIS
LIN {X -103.791,Y 35.1811,Z 112,A 156.604,B 24.9384,C -1.8133,E1 24.8486,E2 289.1953} C_DIS
LIN {X -101.2443,Y 41.9555,Z 112,A 152.8046,B 24.9376,C -1.8244,E1 24.8524,E2 292.9898} C_DIS
LIN {X -97.903,Y 49.2512,Z 112,A 148.6105,B 24.9367,C -1.837,E1 24.8574,E2 297.1765} C_DIS
LIN {X -96.2599,Y 52.3861,Z 112,A 146.7109,B 24.9365,C -1.8407,E1 24.8598,E2 299.0775} C_DIS
LIN {X -93.5158,Y 57.1412,Z 112,A 143.9011,B 24.9358,C -1.8513,E1 24.8638,E2 301.8767} C_DIS
LIN {X -91.9105,Y 59.6895,Z 112,A 141.9929,B 24.9363,C -1.8432,E1 24.8667,E2 303.8138} C_DIS
LIN {X -89.6098,Y 63.0934,Z 112,A 139.9114,B 24.9357,C -1.8516,E1 24.87,E2 305.8854} C_DIS
LIN {X -86.2576,Y 67.6023,Z 112,A 136.2811,B 24.937,C -1.8337,E1 24.8763,E2 309.5759} C_DIS
LIN {X -83.1264,Y 71.4175,Z 112,A 134.5353,B 24.9343,C -1.8717,E1 24.8793,E2 311.2391} C_DIS
LIN {X -78.5895,Y 76.3816,Z 112,A 130.0637,B 24.9362,C -1.8445,E1 24.888,E2 315.7949} C_DIS
LIN {X -74.8184,Y 80.0787,Z 112,A 128.2825,B 24.9332,C -1.888,E1 24.8914,E2 317.4798} C_DIS
LIN {X -70.0191,Y 84.3064,Z 112,A 124.2152,B 24.9346,C -1.8681,E1 24.9001,E2 321.6104} C_DIS
LIN {X -66.816,Y 86.867,Z 112,A 122.6458,B 24.9327,C -1.8945,E1 24.9035,E2 323.1226} C_DIS
LIN {X -63.3058,Y 89.4579,Z 112,A 120.0167,B 24.9333,C -1.8859,E1 24.9095,E2 325.7814} C_DIS
LIN {X -58.9336,Y 92.3969,Z 112,A 117.5908,B 24.932,C -1.9039,E1 24.9151,E2 328.1725} C_DIS
LIN {X -55.8178,Y 94.3114,Z 112,A 115.6707,B 24.9318,C -1.9071,E1 24.9196,E2 330.0909} C_DIS
LIN {X -51.4814,Y 96.7478,Z 112,A 112.5452,B 24.9329,C -1.8913,E1 24.9274,E2 333.2627} C_DIS
LIN {X -48.1356,Y 98.4544,Z 112,A 110.6747,B 24.9325,C -1.8981,E1 24.9321,E2 335.1221} C_DIS
LIN {X -45.083,Y 99.8889,Z 112,A 109.3595,B 24.931,C -1.9181,E1 24.9353,E2 336.3929} C_DIS
LIN {X -42.0004,Y 101.2254,Z 112,A 107.0831,B 24.9323,C -1.9004,E1 24.9413,E2 338.7165} C_DIS
LIN {X -38.7118,Y 102.5264,Z 112,A 105.698,B 24.9308,C -1.921,E1 24.9448,E2 340.0558} C_DIS
LIN {X -35.6943,Y 103.6174,Z 112,A 104.0944,B 24.9305,C -1.926,E1 24.949,E2 341.6506} C_DIS
LIN {X -31.0028,Y 105.1148,Z 112,A 100.9199,B 24.9319,C -1.9055,E1 24.9576,E2 344.8793} C_DIS
LIN {X -27.3205,Y 106.1313,Z 112,A 99.4364,B 24.9303,C -1.9276,E1 24.9615,E2 346.3124} C_DIS
LIN {X -23.6033,Y 107.0196,Z 112,A 96.1557,B 24.9338,C -1.8793,E1 24.9708,E2 349.712} C_DIS
LIN {X -16.7272,Y 108.3072,Z 112,A 94.1756,B 24.9289,C -1.9479,E1 24.9758,E2 351.5309} C_DIS
LIN {X -14.3934,Y 108.6425,Z 112,A 92.468,B 24.9302,C -1.9297,E1 24.9806,E2 353.2831} C_DIS
LIN {X -10.9079,Y 109.0483,Z 112,A 90.6138,B 24.9302,C -1.9299,E1 24.9857,E2 355.138} C_DIS
LIN {X -7.0364,Y 109.3658,Z 112,A 88.713,B 24.9297,C -1.936,E1 24.991,E2 357.025} C_DIS
LIN {X -4.0741,Y 109.5174,Z 112,A 86.985,B 24.9302,C -1.9294,E1 24.9959,E2 358.7692} C_DIS
LIN {X -0.4234,Y 109.5908,Z 112,A 85.1027,B 24.9301,C -1.931,E1 25.0011,E2 360.6478} C_DIS
LIN {X 3.6674,Y 109.5304,Z 112,A 82.969,B 24.9301,C -1.9314,E1 25.0071,E2 362.78} C_DIS
LIN {X 7.7269,Y 109.3191,Z 112,A 80.8513,B 24.9301,C -1.9317,E1 25.013,E2 364.8962} C_DIS
LIN {X 11.6377,Y 108.9719,Z 112,A 78.8127,B 24.9301,C -1.9321,E1 25.0186,E2 366.9327} C_DIS
LIN {X 15.5223,Y 108.4865,Z 112,A 76.8377,B 24.9298,C -1.9345,E1 25.0241,E2 368.9002} C_DIS
LIN {X 20.1575,Y 107.7231,Z 112,A 74.5099,B 24.9295,C -1.9389,E1 25.0304,E2 371.2153} C_DIS
LIN {X 24.1638,Y 106.8954,Z 112,A 71.7746,B 24.9314,C -1.9134,E1 25.0381,E2 374.0074} C_DIS
LIN {X 27.6964,Y 106.0347,Z 112,A 70.2052,B 24.9305,C -1.9258,E1 25.0422,E2 375.5451} C_DIS
LIN {X 31.6586,Y 104.9202,Z 112,A 68.3254,B 24.9298,C -1.9355,E1 25.0472,E2 377.3987} C_DIS
LIN {X 34.4508,Y 104.0373,Z 112,A 65.8325,B 24.9327,C -1.8946,E1 25.0541,E2 379.9836} C_DIS
LIN {X 39.3385,Y 102.2891,Z 112,A 64.0723,B 24.9301,C -1.9314,E1 25.0584,E2 381.653} C_DIS
LIN {X 43.1789,Y 100.7288,Z 112,A 61.7327,B 24.9308,C -1.9219,E1 25.0645,E2 384.0096} C_DIS
LIN {X 48.1729,Y 98.4369,Z 112,A 58.9758,B 24.9307,C -1.9233,E1 25.0714,E2 386.7561} C_DIS
LIN {X 50.4712,Y 97.2793,Z 112,A 56.6985,B 24.9336,C -1.8827,E1 25.0773,E2 389.1232} C_DIS
LIN {X 55.2371,Y 94.6546,Z 112,A 54.8651,B 24.9308,C -1.9208,E1 25.0815,E2 390.8608} C_DIS
LIN {X 58.6259,Y 92.5943,Z 112,A 51.8672,B 24.9338,C -1.8788,E1 25.0888,E2 393.9485} C_DIS
LIN {X 62.8523,Y 89.7774,Z 112,A 50.1775,B 24.9312,C -1.915,E1 25.0925,E2 395.5468} C_DIS
LIN {X 65.0581,Y 88.1921,Z 112,A 48.1547,B 24.9332,C -1.887,E1 25.0972,E2 397.6287} C_DIS
LIN {X 67.9456,Y 85.9864,Z 112,A 46.8261,B 24.9318,C -1.9077,E1 25.1,E2 398.9034} C_DIS
LIN {X 70.2185,Y 84.1407,Z 112,A 45.252,B 24.9321,C -1.903,E1 25.1034,E2 400.4828} C_DIS
LIN {X 73.0258,Y 81.716,Z 112,A 43.2994,B 24.9324,C -1.8985,E1 25.1075,E2 402.438} C_DIS
Enddeposition()
END
